LIN {X 0,Y 564.129,Z 608.975,A -85,B 0,C 180,E1 27064.074,E2 27064.074} C_VEL
LIN {X 0,Y 564.426,Z 588.414,A -85,B 0,C 180,E1 27063.622,E2 27063.622} C_VEL
LIN {X 0,Y 565.706,Z 337.003,A -85,B 0,C 180,E1 27060.121,E2 27060.121} C_VEL
LIN {X 0,Y 564.243,Z 328.893,A -85,B 0,C 180,E1 27059.903,E2 27059.903} C_VEL
LIN {X 0,Y 565.2,Z 283.5,A -85,B 0,C 180,E1 27056.615,E2 27056.615} C_VEL
LIN {X 0,Y 565.283,Z 271.236,A -85,B 0,C 180,E1 27055.692,E2 27055.692} C_VEL
LIN {X 0,Y 560.332,Z 258.325,A -85,B 0,C 180,E1 27054.283,E2 27054.283} C_VEL
LIN {X 0,Y 560.259,Z 257.932,A -85,B 0,C 180,E1 27053.598,E2 27053.598} C_VEL
LIN {X 0,Y 560.276,Z 257.928,A -85,B 0,C 180,E1 27050.278,E2 27050.278} C_VEL
LIN {X 0,Y 560.273,Z 257.936,A -85,B 0,C 180,E1 27047.024,E2 27047.024} C_VEL
LIN {X 0,Y 560.266,Z 257.946,A -85,B 0,C 180,E1 27043.681,E2 27043.681} C_VEL
LIN {X 0,Y 560.273,Z 257.941,A -85,B 0,C 180,E1 27040.359,E2 27040.359} C_VEL
LIN {X 0,Y 560.265,Z 257.937,A -85,B 0,C 180,E1 27036.919,E2 27036.919} C_VEL
LIN {X 0,Y 560.273,Z 257.946,A -85,B 0,C 180,E1 27033.552,E2 27033.552} C_VEL
LIN {X 0,Y 560.267,Z 257.933,A -85,B 0,C 180,E1 27030.216,E2 27030.216} C_VEL
LIN {X 0,Y 560.256,Z 257.943,A -85,B 0,C 180,E1 27026.837,E2 27026.837} C_VEL
LIN {X 0,Y 560.279,Z 257.944,A -85,B 0,C 180,E1 27023.562,E2 27023.562} C_VEL
LIN {X 0,Y 560.246,Z 257.944,A -85,B 0,C 180,E1 27020.366,E2 27020.366} C_VEL
LIN {X 0,Y 560.263,Z 257.948,A -85,B 0,C 180,E1 27017.019,E2 27017.019} C_VEL
LIN {X 0,Y 560.28,Z 257.938,A -85,B 0,C 180,E1 27013.73,E2 27013.73} C_VEL
LIN {X 0,Y 560.233,Z 257.94,A -85,B 0,C 180,E1 27010.469,E2 27010.469} C_VEL
LIN {X 0,Y 560.274,Z 257.945,A -85,B 0,C 180,E1 27007.176,E2 27007.176} C_VEL
LIN {X 0,Y 560.24,Z 257.945,A -85,B 0,C 180,E1 27003.957,E2 27003.957} C_VEL
LIN {X 0,Y 560.224,Z 257.947,A -85,B 0,C 180,E1 27000.614,E2 27000.614} C_VEL
LIN {X 0,Y 560.278,Z 257.945,A -85,B 0,C 180,E1 26997.443,E2 26997.443} C_VEL
LIN {X 0,Y 560.21,Z 257.947,A -85,B 0,C 180,E1 26994.264,E2 26994.264} C_VEL
LIN {X 0,Y 560.256,Z 257.949,A -85,B 0,C 180,E1 26991.068,E2 26991.068} C_VEL
LIN {X 0,Y 560.209,Z 257.945,A -85,B 0,C 180,E1 26987.947,E2 26987.947} C_VEL
LIN {X 0,Y 560.203,Z 257.945,A -85,B 0,C 180,E1 26984.53,E2 26984.53} C_VEL
LIN {X 0,Y 560.246,Z 257.949,A -85,B 0,C 180,E1 26981.478,E2 26981.478} C_VEL
LIN {X 0,Y 560.206,Z 257.948,A -85,B 0,C 180,E1 26978.318,E2 26978.318} C_VEL
LIN {X 0,Y 560.277,Z 257.949,A -85,B 0,C 180,E1 26975.205,E2 26975.205} C_VEL
LIN {X 0,Y 560.214,Z 257.948,A -85,B 0,C 180,E1 26972.005,E2 26972.005} C_VEL
LIN {X 0,Y 560.248,Z 257.935,A -85,B 0,C 180,E1 26968.712,E2 26968.712} C_VEL
LIN {X 0,Y 560.249,Z 257.949,A -85,B 0,C 180,E1 26965.537,E2 26965.537} C_VEL
LIN {X 0,Y 560.229,Z 257.942,A -85,B 0,C 180,E1 26962.243,E2 26962.243} C_VEL
LIN {X 0,Y 560.283,Z 257.933,A -85,B 0,C 180,E1 26959.012,E2 26959.012} C_VEL
LIN {X 0,Y 560.241,Z 257.949,A -85,B 0,C 180,E1 26955.748,E2 26955.748} C_VEL
LIN {X 0,Y 560.252,Z 257.945,A -85,B 0,C 180,E1 26952.367,E2 26952.367} C_VEL
LIN {X 0,Y 560.281,Z 257.941,A -85,B 0,C 180,E1 26949.079,E2 26949.079} C_VEL
LIN {X 0,Y 560.319,Z 258.259,A -85,B 0,C 180,E1 26948.567,E2 26948.567} C_VEL
LIN {X 0,Y 564.336,Z 267.794,A -85,B 0,C 180,E1 26947.551,E2 26947.551} C_VEL
LIN {X 0,Y 566.828,Z 273.642,A -85,B 0,C 180,E1 26946.959,E2 26946.959} C_VEL
LIN {X 0,Y 566.291,Z 302.779,A -85,B 0,C 180,E1 26945.075,E2 26945.075} C_VEL
LIN {X 0,Y 567.756,Z 312.242,A -85,B 0,C 180,E1 26944.825,E2 26944.825} C_VEL
LIN {X 0,Y 566.415,Z 533.81,A -85,B 0,C 180,E1 26941.628,E2 26941.628} C_VEL
LIN {X 0,Y 565.943,Z 609.207,A -85,B 0,C 180,E1 26940.529,E2 26940.529} C_VEL
LIN {X 0,Y 565.546,Z 630.675,A -85,B 0,C 180,E1 26940.025,E2 26940.025} C_VEL
LIN {X 0,Y 565.085,Z 652.51,A -85,B 0,C 180,E1 26939.319,E2 26939.319} C_VEL
LIN {X 0,Y 564.579,Z 673.407,A -85,B 0,C 180,E1 26938.449,E2 26938.449} C_VEL
LIN {X 0,Y 563.935,Z 693.757,A -85,B 0,C 180,E1 26937.392,E2 26937.392} C_VEL
LIN {X 0,Y 563.301,Z 714.152,A -85,B 0,C 180,E1 26936.116,E2 26936.116} C_VEL
LIN {X 0,Y 562.7,Z 732.379,A -85,B 0,C 180,E1 26934.771,E2 26934.771} C_VEL
LIN {X 0,Y 562.102,Z 750.23,A -85,B 0,C 180,E1 26933.229,E2 26933.229} C_VEL
LIN {X 0,Y 561.572,Z 766.692,A -85,B 0,C 180,E1 26931.571,E2 26931.571} C_VEL
LIN {X 0,Y 561.082,Z 782.874,A -85,B 0,C 180,E1 26929.682,E2 26929.682} C_VEL
LIN {X 0,Y 560.714,Z 797.045,A -85,B 0,C 180,E1 26927.753,E2 26927.753} C_VEL
LIN {X 0,Y 560.417,Z 809.739,A -85,B 0,C 180,E1 26925.735,E2 26925.735} C_VEL
LIN {X 0,Y 560.198,Z 820.334,A -85,B 0,C 180,E1 26923.732,E2 26923.732} C_VEL
LIN {X 0,Y 560.057,Z 830.069,A -85,B 0,C 180,E1 26921.534,E2 26921.534} C_VEL
LIN {X 0,Y 559.982,Z 837.937,A -85,B 0,C 180,E1 26919.351,E2 26919.351} C_VEL
LIN {X 0,Y 559.938,Z 843.907,A -85,B 0,C 180,E1 26917.18,E2 26917.18} C_VEL
LIN {X 0,Y 559.917,Z 848.581,A -85,B 0,C 180,E1 26914.841,E2 26914.841} C_VEL
LIN {X 0,Y 559.907,Z 851.338,A -85,B 0,C 180,E1 26912.661,E2 26912.661} C_VEL
LIN {X 0,Y 559.896,Z 852.395,A -85,B 0,C 180,E1 26910.512,E2 26910.512} C_VEL
LIN {X 0,Y 559.901,Z 851.948,A -85,B 0,C 180,E1 26908.26,E2 26908.26} C_VEL
LIN {X 0,Y 559.908,Z 849.994,A -85,B 0,C 180,E1 26906.109,E2 26906.109} C_VEL
LIN {X 0,Y 559.921,Z 846.398,A -85,B 0,C 180,E1 26903.952,E2 26903.952} C_VEL
LIN {X 0,Y 559.958,Z 841.281,A -85,B 0,C 180,E1 26901.788,E2 26901.788} C_VEL
LIN {X 0,Y 560.01,Z 834.757,A -85,B 0,C 180,E1 26899.715,E2 26899.715} C_VEL
LIN {X 0,Y 560.11,Z 826.141,A -85,B 0,C 180,E1 26897.526,E2 26897.526} C_VEL
LIN {X 0,Y 560.286,Z 816.122,A -85,B 0,C 180,E1 26895.427,E2 26895.427} C_VEL
LIN {X 0,Y 560.527,Z 804.629,A -85,B 0,C 180,E1 26893.417,E2 26893.417} C_VEL
LIN {X 0,Y 560.838,Z 791.792,A -85,B 0,C 180,E1 26891.499,E2 26891.499} C_VEL
LIN {X 0,Y 561.233,Z 777.662,A -85,B 0,C 180,E1 26889.672,E2 26889.672} C_VEL
LIN {X 0,Y 561.73,Z 761.816,A -85,B 0,C 180,E1 26887.907,E2 26887.907} C_VEL
LIN {X 0,Y 562.275,Z 745.074,A -85,B 0,C 180,E1 26886.305,E2 26886.305} C_VEL
LIN {X 0,Y 562.893,Z 726.402,A -85,B 0,C 180,E1 26884.767,E2 26884.767} C_VEL
LIN {X 0,Y 563.512,Z 707.543,A -85,B 0,C 180,E1 26883.441,E2 26883.441} C_VEL
LIN {X 0,Y 564.132,Z 687.761,A -85,B 0,C 180,E1 26882.274,E2 26882.274} C_VEL
LIN {X 0,Y 564.706,Z 667.063,A -85,B 0,C 180,E1 26881.269,E2 26881.269} C_VEL
LIN {X 0,Y 565.266,Z 645.686,A -85,B 0,C 180,E1 26880.438,E2 26880.438} C_VEL
LIN {X 0,Y 565.67,Z 624.869,A -85,B 0,C 180,E1 26879.819,E2 26879.819} C_VEL
LIN {X 0,Y 565.988,Z 603.285,A -85,B 0,C 180,E1 26879.372,E2 26879.372} C_VEL
LIN {X 0,Y 567.374,Z 374.728,A -85,B 0,C 180,E1 26876.087,E2 26876.087} C_VEL
LIN {X 0,Y 567.577,Z 309.911,A -85,B 0,C 180,E1 26875.127,E2 26875.127} C_VEL
LIN {X 0,Y 566.208,Z 301.853,A -85,B 0,C 180,E1 26874.885,E2 26874.885} C_VEL
LIN {X 0,Y 566.754,Z 273.379,A -85,B 0,C 180,E1 26873.018,E2 26873.018} C_VEL
LIN {X 0,Y 560.335,Z 258.355,A -85,B 0,C 180,E1 26871.451,E2 26871.451} C_VEL
LIN {X 0,Y 560.279,Z 257.933,A -85,B 0,C 180,E1 26871.084,E2 26871.084} C_VEL
LIN {X 0,Y 560.242,Z 257.947,A -85,B 0,C 180,E1 26867.854,E2 26867.854} C_VEL
LIN {X 0,Y 560.254,Z 257.947,A -85,B 0,C 180,E1 26864.452,E2 26864.452} C_VEL
LIN {X 0,Y 560.283,Z 257.932,A -85,B 0,C 180,E1 26861.144,E2 26861.144} C_VEL
LIN {X 0,Y 560.228,Z 257.942,A -85,B 0,C 180,E1 26857.875,E2 26857.875} C_VEL
LIN {X 0,Y 560.263,Z 257.949,A -85,B 0,C 180,E1 26854.577,E2 26854.577} C_VEL
LIN {X 0,Y 560.237,Z 257.936,A -85,B 0,C 180,E1 26851.408,E2 26851.408} C_VEL
LIN {X 0,Y 560.221,Z 257.948,A -85,B 0,C 180,E1 26848.11,E2 26848.11} C_VEL
LIN {X 0,Y 560.272,Z 257.945,A -85,B 0,C 180,E1 26844.967,E2 26844.967} C_VEL
LIN {X 0,Y 560.207,Z 257.948,A -85,B 0,C 180,E1 26841.792,E2 26841.792} C_VEL
LIN {X 0,Y 560.265,Z 257.948,A -85,B 0,C 180,E1 26838.629,E2 26838.629} C_VEL
LIN {X 0,Y 560.2,Z 257.945,A -85,B 0,C 180,E1 26835.529,E2 26835.529} C_VEL
LIN {X 0,Y 560.213,Z 257.945,A -85,B 0,C 180,E1 26832.158,E2 26832.158} C_VEL
LIN {X 0,Y 560.228,Z 257.949,A -85,B 0,C 180,E1 26829.139,E2 26829.139} C_VEL
LIN {X 0,Y 560.209,Z 257.948,A -85,B 0,C 180,E1 26825.839,E2 26825.839} C_VEL
LIN {X 0,Y 560.278,Z 257.944,A -85,B 0,C 180,E1 26822.659,E2 26822.659} C_VEL
LIN {X 0,Y 560.216,Z 257.947,A -85,B 0,C 180,E1 26819.488,E2 26819.488} C_VEL
LIN {X 0,Y 560.255,Z 257.944,A -85,B 0,C 180,E1 26816.214,E2 26816.214} C_VEL
LIN {X 0,Y 560.247,Z 257.944,A -85,B 0,C 180,E1 26813.029,E2 26813.029} C_VEL
LIN {X 0,Y 560.23,Z 257.94,A -85,B 0,C 180,E1 26809.719,E2 26809.719} C_VEL
LIN {X 0,Y 560.284,Z 257.941,A -85,B 0,C 180,E1 26806.48,E2 26806.48} C_VEL
LIN {X 0,Y 560.238,Z 257.946,A -85,B 0,C 180,E1 26803.301,E2 26803.301} C_VEL
LIN {X 0,Y 560.262,Z 257.942,A -85,B 0,C 180,E1 26799.961,E2 26799.961} C_VEL
LIN {X 0,Y 560.28,Z 257.946,A -85,B 0,C 180,E1 26796.661,E2 26796.661} C_VEL
LIN {X 0,Y 560.28,Z 257.942,A -85,B 0,C 180,E1 26796.239,E2 26796.239} C_VEL
LIN {X 0,Y 559.29,Z 258.064,A -85,B 0,C 180,E1 26795.451,E2 26795.451} C_VEL
LIN {X 0,Y 552.863,Z 258.863,A -85,B 0,C 180,E1 26793.24,E2 26793.24} C_VEL
LIN {X 0,Y 552.339,Z 258.936,A -85,B 0,C 180,E1 26792.664,E2 26792.664} C_VEL
LIN {X 0,Y 552.312,Z 258.925,A -85,B 0,C 180,E1 26789.302,E2 26789.302} C_VEL
LIN {X 0,Y 552.339,Z 258.93,A -85,B 0,C 180,E1 26785.988,E2 26785.988} C_VEL
LIN {X 0,Y 552.336,Z 258.922,A -85,B 0,C 180,E1 26782.537,E2 26782.537} C_VEL
LIN {X 0,Y 552.321,Z 258.934,A -85,B 0,C 180,E1 26779.193,E2 26779.193} C_VEL
LIN {X 0,Y 552.342,Z 258.93,A -85,B 0,C 180,E1 26775.793,E2 26775.793} C_VEL
LIN {X 0,Y 552.33,Z 258.93,A -85,B 0,C 180,E1 26772.389,E2 26772.389} C_VEL
LIN {X 0,Y 552.328,Z 258.921,A -85,B 0,C 180,E1 26769.18,E2 26769.18} C_VEL
LIN {X 0,Y 552.355,Z 259.158,A -85,B 0,C 180,E1 26766.207,E2 26766.207} C_VEL
LIN {X 0,Y 554.368,Z 264.541,A -85,B 0,C 180,E1 26765.568,E2 26765.568} C_VEL
LIN {X 0,Y 558.48,Z 275.126,A -85,B 0,C 180,E1 26764.413,E2 26764.413} C_VEL
LIN {X 0,Y 557.294,Z 318.934,A -85,B 0,C 180,E1 26761.151,E2 26761.151} C_VEL
LIN {X 0,Y 557.128,Z 329.515,A -85,B 0,C 180,E1 26760.412,E2 26760.412} C_VEL
LIN {X 0,Y 558.767,Z 339.665,A -85,B 0,C 180,E1 26760.159,E2 26760.159} C_VEL
LIN {X 0,Y 557.241,Z 590.093,A -85,B 0,C 180,E1 26756.626,E2 26756.626} C_VEL
LIN {X 0,Y 556.889,Z 610.371,A -85,B 0,C 180,E1 26756.16,E2 26756.16} C_VEL
LIN {X 0,Y 556.454,Z 630.143,A -85,B 0,C 180,E1 26755.517,E2 26755.517} C_VEL
LIN {X 0,Y 555.93,Z 650.229,A -85,B 0,C 180,E1 26754.661,E2 26754.661} C_VEL
LIN {X 0,Y 555.374,Z 668.831,A -85,B 0,C 180,E1 26753.67,E2 26753.67} C_VEL
LIN {X 0,Y 554.772,Z 687.426,A -85,B 0,C 180,E1 26752.462,E2 26752.462} C_VEL
LIN {X 0,Y 554.193,Z 704.475,A -85,B 0,C 180,E1 26751.131,E2 26751.131} C_VEL
LIN {X 0,Y 553.647,Z 720.769,A -85,B 0,C 180,E1 26749.627,E2 26749.627} C_VEL
LIN {X 0,Y 553.165,Z 735.716,A -85,B 0,C 180,E1 26748.004,E2 26748.004} C_VEL
LIN {X 0,Y 552.773,Z 749.225,A -85,B 0,C 180,E1 26746.282,E2 26746.282} C_VEL
LIN {X 0,Y 552.443,Z 761.975,A -85,B 0,C 180,E1 26744.356,E2 26744.356} C_VEL
LIN {X 0,Y 552.224,Z 772.578,A -85,B 0,C 180,E1 26742.442,E2 26742.442} C_VEL
LIN {X 0,Y 552.074,Z 781.763,A -85,B 0,C 180,E1 26740.434,E2 26740.434} C_VEL
LIN {X 0,Y 551.983,Z 789.382,A -85,B 0,C 180,E1 26738.332,E2 26738.332} C_VEL
LIN {X 0,Y 551.934,Z 794.889,A -85,B 0,C 180,E1 26736.344,E2 26736.344} C_VEL
LIN {X 0,Y 551.917,Z 799.202,A -85,B 0,C 180,E1 26734.155,E2 26734.155} C_VEL
LIN {X 0,Y 551.914,Z 801.641,A -85,B 0,C 180,E1 26732.076,E2 26732.076} C_VEL
LIN {X 0,Y 551.914,Z 802.495,A -85,B 0,C 180,E1 26730,E2 26730} C_VEL
LIN {X 0,Y 551.909,Z 801.633,A -85,B 0,C 180,E1 26727.82,E2 26727.82} C_VEL
LIN {X 0,Y 551.914,Z 799.18,A -85,B 0,C 180,E1 26725.74,E2 26725.74} C_VEL
LIN {X 0,Y 551.932,Z 794.854,A -85,B 0,C 180,E1 26723.551,E2 26723.551} C_VEL
LIN {X 0,Y 551.983,Z 788.979,A -85,B 0,C 180,E1 26721.458,E2 26721.458} C_VEL
LIN {X 0,Y 552.075,Z 781.702,A -85,B 0,C 180,E1 26719.46,E2 26719.46} C_VEL
LIN {X 0,Y 552.228,Z 772.238,A -85,B 0,C 180,E1 26717.398,E2 26717.398} C_VEL
LIN {X 0,Y 552.451,Z 761.83,A -85,B 0,C 180,E1 26715.53,E2 26715.53} C_VEL
LIN {X 0,Y 552.774,Z 749.093,A -85,B 0,C 180,E1 26713.611,E2 26713.611} C_VEL
LIN {X 0,Y 553.196,Z 734.628,A -85,B 0,C 180,E1 26711.779,E2 26711.779} C_VEL
LIN {X 0,Y 553.707,Z 718.916,A -85,B 0,C 180,E1 26710.1,E2 26710.1} C_VEL
LIN {X 0,Y 554.284,Z 701.829,A -85,B 0,C 180,E1 26708.56,E2 26708.56} C_VEL
LIN {X 0,Y 554.885,Z 683.925,A -85,B 0,C 180,E1 26707.207,E2 26707.207} C_VEL
LIN {X 0,Y 555.472,Z 665.466,A -85,B 0,C 180,E1 26706.045,E2 26706.045} C_VEL
LIN {X 0,Y 556.05,Z 646.345,A -85,B 0,C 180,E1 26705.061,E2 26705.061} C_VEL
LIN {X 0,Y 556.56,Z 626.554,A -85,B 0,C 180,E1 26704.26,E2 26704.26} C_VEL
LIN {X 0,Y 556.951,Z 606.601,A -85,B 0,C 180,E1 26703.65,E2 26703.65} C_VEL
LIN {X 0,Y 557.269,Z 585.492,A -85,B 0,C 180,E1 26703.208,E2 26703.208} C_VEL
LIN {X 0,Y 558.743,Z 338.271,A -85,B 0,C 180,E1 26699.729,E2 26699.729} C_VEL
LIN {X 0,Y 557.057,Z 328.892,A -85,B 0,C 180,E1 26699.473,E2 26699.473} C_VEL
LIN {X 0,Y 558.187,Z 284.604,A -85,B 0,C 180,E1 26696.217,E2 26696.217} C_VEL
LIN {X 0,Y 558.38,Z 274.72,A -85,B 0,C 180,E1 26695.457,E2 26695.457} C_VEL
LIN {X 0,Y 552.364,Z 259.241,A -85,B 0,C 180,E1 26693.724,E2 26693.724} C_VEL
LIN {X 0,Y 552.336,Z 258.926,A -85,B 0,C 180,E1 26692.627,E2 26692.627} C_VEL
LIN {X 0,Y 552.343,Z 258.929,A -85,B 0,C 180,E1 26689.172,E2 26689.172} C_VEL
LIN {X 0,Y 552.325,Z 258.925,A -85,B 0,C 180,E1 26685.797,E2 26685.797} C_VEL
LIN {X 0,Y 552.329,Z 258.916,A -85,B 0,C 180,E1 26682.472,E2 26682.472} C_VEL
LIN {X 0,Y 552.334,Z 258.931,A -85,B 0,C 180,E1 26679.048,E2 26679.048} C_VEL
LIN {X 0,Y 552.333,Z 258.927,A -85,B 0,C 180,E1 26675.632,E2 26675.632} C_VEL
LIN {X 0,Y 552.328,Z 258.923,A -85,B 0,C 180,E1 26672.278,E2 26672.278} C_VEL
LIN {X 0,Y 552.319,Z 258.935,A -85,B 0,C 180,E1 26668.818,E2 26668.818} C_VEL
LIN {X 0,Y 552.339,Z 258.93,A -85,B 0,C 180,E1 26665.521,E2 26665.521} C_VEL
LIN {X 0,Y 552.316,Z 258.927,A -85,B 0,C 180,E1 26662.232,E2 26662.232} C_VEL
LIN {X 0,Y 552.309,Z 258.932,A -85,B 0,C 180,E1 26658.778,E2 26658.778} C_VEL
LIN {X 0,Y 552.345,Z 258.934,A -85,B 0,C 180,E1 26655.433,E2 26655.433} C_VEL
LIN {X 0,Y 552.306,Z 258.933,A -85,B 0,C 180,E1 26652.122,E2 26652.122} C_VEL
LIN {X 0,Y 552.298,Z 258.936,A -85,B 0,C 180,E1 26648.725,E2 26648.725} C_VEL
LIN {X 0,Y 552.343,Z 258.929,A -85,B 0,C 180,E1 26645.506,E2 26645.506} C_VEL
LIN {X 0,Y 552.284,Z 258.933,A -85,B 0,C 180,E1 26642.283,E2 26642.283} C_VEL
LIN {X 0,Y 552.31,Z 258.936,A -85,B 0,C 180,E1 26638.963,E2 26638.963} C_VEL
LIN {X 0,Y 552.294,Z 258.934,A -85,B 0,C 180,E1 26635.847,E2 26635.847} C_VEL
LIN {X 0,Y 552.272,Z 258.934,A -85,B 0,C 180,E1 26632.51,E2 26632.51} C_VEL
LIN {X 0,Y 552.33,Z 258.936,A -85,B 0,C 180,E1 26629.36,E2 26629.36} C_VEL
LIN {X 0,Y 552.26,Z 258.938,A -85,B 0,C 180,E1 26626.174,E2 26626.174} C_VEL
LIN {X 0,Y 552.296,Z 258.938,A -85,B 0,C 180,E1 26622.91,E2 26622.91} C_VEL
LIN {X 0,Y 552.279,Z 258.935,A -85,B 0,C 180,E1 26619.77,E2 26619.77} C_VEL
LIN {X 0,Y 552.273,Z 258.935,A -85,B 0,C 180,E1 26616.415,E2 26616.415} C_VEL
LIN {X 0,Y 552.342,Z 258.933,A -85,B 0,C 180,E1 26613.178,E2 26613.178} C_VEL
LIN {X 0,Y 552.279,Z 258.933,A -85,B 0,C 180,E1 26610.022,E2 26610.022} C_VEL
LIN {X 0,Y 552.317,Z 258.935,A -85,B 0,C 180,E1 26606.735,E2 26606.735} C_VEL
LIN {X 0,Y 552.306,Z 258.928,A -85,B 0,C 180,E1 26603.574,E2 26603.574} C_VEL
LIN {X 0,Y 552.296,Z 258.935,A -85,B 0,C 180,E1 26600.279,E2 26600.279} C_VEL
LIN {X 0,Y 552.345,Z 258.934,A -85,B 0,C 180,E1 26596.996,E2 26596.996} C_VEL
LIN {X 0,Y 552.302,Z 258.927,A -85,B 0,C 180,E1 26593.752,E2 26593.752} C_VEL
LIN {X 0,Y 552.314,Z 258.924,A -85,B 0,C 180,E1 26590.347,E2 26590.347} C_VEL
LIN {X 0,Y 552.38,Z 259.179,A -85,B 0,C 180,E1 26589.176,E2 26589.176} C_VEL
LIN {X 0,Y 554.318,Z 264.07,A -85,B 0,C 180,E1 26588.615,E2 26588.615} C_VEL
LIN {X 0,Y 560.022,Z 277.103,A -85,B 0,C 180,E1 26587.245,E2 26587.245} C_VEL
LIN {X 0,Y 559.467,Z 302.819,A -85,B 0,C 180,E1 26585.567,E2 26585.567} C_VEL
LIN {X 0,Y 561.178,Z 313.62,A -85,B 0,C 180,E1 26585.273,E2 26585.273} C_VEL
LIN {X 0,Y 559.597,Z 534.701,A -85,B 0,C 180,E1 26582.046,E2 26582.046} C_VEL
LIN {X 0,Y 559.047,Z 609.207,A -85,B 0,C 180,E1 26580.946,E2 26580.946} C_VEL
LIN {X 0,Y 558.581,Z 630.676,A -85,B 0,C 180,E1 26580.438,E2 26580.438} C_VEL
LIN {X 0,Y 558.051,Z 652.58,A -85,B 0,C 180,E1 26579.722,E2 26579.722} C_VEL
LIN {X 0,Y 557.44,Z 673.407,A -85,B 0,C 180,E1 26578.848,E2 26578.848} C_VEL
LIN {X 0,Y 556.703,Z 693.759,A -85,B 0,C 180,E1 26577.779,E2 26577.779} C_VEL
LIN {X 0,Y 555.951,Z 714.153,A -85,B 0,C 180,E1 26576.488,E2 26576.488} C_VEL
LIN {X 0,Y 555.199,Z 733.16,A -85,B 0,C 180,E1 26575.062,E2 26575.062} C_VEL
LIN {X 0,Y 554.505,Z 751.116,A -85,B 0,C 180,E1 26573.484,E2 26573.484} C_VEL
LIN {X 0,Y 553.868,Z 767.704,A -85,B 0,C 180,E1 26571.775,E2 26571.775} C_VEL
LIN {X 0,Y 553.323,Z 782.875,A -85,B 0,C 180,E1 26569.969,E2 26569.969} C_VEL
LIN {X 0,Y 552.873,Z 797.046,A -85,B 0,C 180,E1 26568.013,E2 26568.013} C_VEL
LIN {X 0,Y 552.515,Z 809.737,A -85,B 0,C 180,E1 26565.966,E2 26565.966} C_VEL
LIN {X 0,Y 552.258,Z 820.335,A -85,B 0,C 180,E1 26563.933,E2 26563.933} C_VEL
LIN {X 0,Y 552.085,Z 830.07,A -85,B 0,C 180,E1 26561.703,E2 26561.703} C_VEL
LIN {X 0,Y 551.99,Z 837.937,A -85,B 0,C 180,E1 26559.487,E2 26559.487} C_VEL
LIN {X 0,Y 551.939,Z 843.908,A -85,B 0,C 180,E1 26557.285,E2 26557.285} C_VEL
LIN {X 0,Y 551.92,Z 848.464,A -85,B 0,C 180,E1 26554.988,E2 26554.988} C_VEL
LIN {X 0,Y 551.909,Z 851.234,A -85,B 0,C 180,E1 26552.804,E2 26552.804} C_VEL
LIN {X 0,Y 551.898,Z 852.373,A -85,B 0,C 180,E1 26550.623,E2 26550.623} C_VEL
LIN {X 0,Y 551.899,Z 852.015,A -85,B 0,C 180,E1 26548.339,E2 26548.339} C_VEL
LIN {X 0,Y 551.904,Z 850.221,A -85,B 0,C 180,E1 26546.261,E2 26546.261} C_VEL
LIN {X 0,Y 551.922,Z 846.603,A -85,B 0,C 180,E1 26543.969,E2 26543.969} C_VEL
LIN {X 0,Y 551.965,Z 841.584,A -85,B 0,C 180,E1 26541.773,E2 26541.773} C_VEL
LIN {X 0,Y 552.025,Z 835.112,A -85,B 0,C 180,E1 26539.67,E2 26539.67} C_VEL
LIN {X 0,Y 552.147,Z 826.537,A -85,B 0,C 180,E1 26537.434,E2 26537.434} C_VEL
LIN {X 0,Y 552.351,Z 816.69,A -85,B 0,C 180,E1 26535.32,E2 26535.32} C_VEL
LIN {X 0,Y 552.633,Z 805.272,A -85,B 0,C 180,E1 26533.282,E2 26533.282} C_VEL
LIN {X 0,Y 553.028,Z 791.794,A -85,B 0,C 180,E1 26531.228,E2 26531.228} C_VEL
LIN {X 0,Y 553.514,Z 777.375,A -85,B 0,C 180,E1 26529.342,E2 26529.342} C_VEL
LIN {X 0,Y 554.097,Z 761.625,A -85,B 0,C 180,E1 26527.565,E2 26527.565} C_VEL
LIN {X 0,Y 554.754,Z 744.464,A -85,B 0,C 180,E1 26525.907,E2 26525.907} C_VEL
LIN {X 0,Y 555.498,Z 725.678,A -85,B 0,C 180,E1 26524.35,E2 26524.35} C_VEL
LIN {X 0,Y 556.241,Z 706.421,A -85,B 0,C 180,E1 26522.993,E2 26522.993} C_VEL
LIN {X 0,Y 556.971,Z 686.522,A -85,B 0,C 180,E1 26521.815,E2 26521.815} C_VEL
LIN {X 0,Y 557.64,Z 666.234,A -85,B 0,C 180,E1 26520.832,E2 26520.832} C_VEL
LIN {X 0,Y 558.264,Z 644.481,A -85,B 0,C 180,E1 26519.988,E2 26519.988} C_VEL
LIN {X 0,Y 558.791,Z 623.167,A -85,B 0,C 180,E1 26519.36,E2 26519.36} C_VEL
LIN {X 0,Y 559.113,Z 601.498,A -85,B 0,C 180,E1 26518.923,E2 26518.923} C_VEL
LIN {X 0,Y 560.716,Z 377.149,A -85,B 0,C 180,E1 26515.665,E2 26515.665} C_VEL
LIN {X 0,Y 561.004,Z 311.391,A -85,B 0,C 180,E1 26514.68,E2 26514.68} C_VEL
LIN {X 0,Y 559.388,Z 302.303,A -85,B 0,C 180,E1 26514.417,E2 26514.417} C_VEL
LIN {X 0,Y 559.891,Z 276.6,A -85,B 0,C 180,E1 26512.71,E2 26512.71} C_VEL
LIN {X 0,Y 552.401,Z 259.313,A -85,B 0,C 180,E1 26510.854,E2 26510.854} C_VEL
LIN {X 0,Y 552.309,Z 258.936,A -85,B 0,C 180,E1 26510.281,E2 26510.281} C_VEL
LIN {X 0,Y 552.343,Z 258.935,A -85,B 0,C 180,E1 26506.966,E2 26506.966} C_VEL
LIN {X 0,Y 552.302,Z 258.936,A -85,B 0,C 180,E1 26503.753,E2 26503.753} C_VEL
LIN {X 0,Y 552.306,Z 258.937,A -85,B 0,C 180,E1 26500.348,E2 26500.348} C_VEL
LIN {X 0,Y 552.343,Z 258.922,A -85,B 0,C 180,E1 26497.07,E2 26497.07} C_VEL
LIN {X 0,Y 552.286,Z 258.936,A -85,B 0,C 180,E1 26493.804,E2 26493.804} C_VEL
LIN {X 0,Y 552.308,Z 258.929,A -85,B 0,C 180,E1 26490.457,E2 26490.457} C_VEL
LIN {X 0,Y 552.295,Z 258.936,A -85,B 0,C 180,E1 26487.376,E2 26487.376} C_VEL
LIN {X 0,Y 552.274,Z 258.936,A -85,B 0,C 180,E1 26484.038,E2 26484.038} C_VEL
LIN {X 0,Y 552.334,Z 258.936,A -85,B 0,C 180,E1 26480.892,E2 26480.892} C_VEL
LIN {X 0,Y 552.261,Z 258.938,A -85,B 0,C 180,E1 26477.707,E2 26477.707} C_VEL
LIN {X 0,Y 552.303,Z 258.938,A -85,B 0,C 180,E1 26474.467,E2 26474.467} C_VEL
LIN {X 0,Y 552.268,Z 258.934,A -85,B 0,C 180,E1 26471.381,E2 26471.381} C_VEL
LIN {X 0,Y 552.273,Z 258.934,A -85,B 0,C 180,E1 26467.993,E2 26467.993} C_VEL
LIN {X 0,Y 552.32,Z 258.938,A -85,B 0,C 180,E1 26464.881,E2 26464.881} C_VEL
LIN {X 0,Y 552.273,Z 258.935,A -85,B 0,C 180,E1 26461.66,E2 26461.66} C_VEL
LIN {X 0,Y 552.337,Z 258.931,A -85,B 0,C 180,E1 26458.444,E2 26458.444} C_VEL
LIN {X 0,Y 552.293,Z 258.937,A -85,B 0,C 180,E1 26455.223,E2 26455.223} C_VEL
LIN {X 0,Y 552.292,Z 258.934,A -85,B 0,C 180,E1 26451.777,E2 26451.777} C_VEL
LIN {X 0,Y 552.344,Z 258.935,A -85,B 0,C 180,E1 26448.514,E2 26448.514} C_VEL
LIN {X 0,Y 552.3,Z 258.932,A -85,B 0,C 180,E1 26445.211,E2 26445.211} C_VEL
LIN {X 0,Y 552.306,Z 258.929,A -85,B 0,C 180,E1 26441.748,E2 26441.748} C_VEL
LIN {X 0,Y 552.342,Z 258.93,A -85,B 0,C 180,E1 26438.44,E2 26438.44} C_VEL
LIN {X 0,Y 552.315,Z 258.936,A -85,B 0,C 180,E1 26435.085,E2 26435.085} C_VEL
LIN {X 0,Y 552.339,Z 258.936,A -85,B 0,C 180,E1 26432.664,E2 26432.664} C_VEL
LIN {X 0,Y 551.351,Z 259.069,A -85,B 0,C 180,E1 26431.865,E2 26431.865} C_VEL
LIN {X 0,Y 544.892,Z 259.852,A -85,B 0,C 180,E1 26429.621,E2 26429.621} C_VEL
LIN {X 0,Y 544.381,Z 259.909,A -85,B 0,C 180,E1 26429.036,E2 26429.036} C_VEL
LIN {X 0,Y 544.383,Z 259.921,A -85,B 0,C 180,E1 26425.549,E2 26425.549} C_VEL
LIN {X 0,Y 544.397,Z 259.911,A -85,B 0,C 180,E1 26422.16,E2 26422.16} C_VEL
LIN {X 0,Y 544.403,Z 259.913,A -85,B 0,C 180,E1 26418.69,E2 26418.69} C_VEL
LIN {X 0,Y 544.387,Z 259.923,A -85,B 0,C 180,E1 26415.296,E2 26415.296} C_VEL
LIN {X 0,Y 544.392,Z 259.923,A -85,B 0,C 180,E1 26411.94,E2 26411.94} C_VEL
LIN {X 0,Y 544.393,Z 259.918,A -85,B 0,C 180,E1 26408.507,E2 26408.507} C_VEL
LIN {X 0,Y 544.429,Z 260.124,A -85,B 0,C 180,E1 26406.776,E2 26406.776} C_VEL
LIN {X 0,Y 546.9,Z 266.49,A -85,B 0,C 180,E1 26406.002,E2 26406.002} C_VEL
LIN {X 0,Y 551.518,Z 278.593,A -85,B 0,C 180,E1 26404.663,E2 26404.663} C_VEL
LIN {X 0,Y 550.088,Z 321.904,A -85,B 0,C 180,E1 26401.382,E2 26401.382} C_VEL
LIN {X 0,Y 549.978,Z 329.548,A -85,B 0,C 180,E1 26400.851,E2 26400.851} C_VEL
LIN {X 0,Y 551.844,Z 341.053,A -85,B 0,C 180,E1 26400.558,E2 26400.558} C_VEL
LIN {X 0,Y 550.091,Z 589.816,A -85,B 0,C 180,E1 26397.006,E2 26397.006} C_VEL
LIN {X 0,Y 549.687,Z 610.241,A -85,B 0,C 180,E1 26396.533,E2 26396.533} C_VEL
LIN {X 0,Y 549.193,Z 630.159,A -85,B 0,C 180,E1 26395.879,E2 26395.879} C_VEL
LIN {X 0,Y 548.585,Z 650.241,A -85,B 0,C 180,E1 26395.014,E2 26395.014} C_VEL
LIN {X 0,Y 547.939,Z 668.839,A -85,B 0,C 180,E1 26394.011,E2 26394.011} C_VEL
LIN {X 0,Y 547.252,Z 687.434,A -85,B 0,C 180,E1 26392.788,E2 26392.788} C_VEL
LIN {X 0,Y 546.545,Z 705.568,A -85,B 0,C 180,E1 26391.349,E2 26391.349} C_VEL
LIN {X 0,Y 545.91,Z 721.881,A -85,B 0,C 180,E1 26389.805,E2 26389.805} C_VEL
LIN {X 0,Y 545.354,Z 736.646,A -85,B 0,C 180,E1 26388.16,E2 26388.16} C_VEL
LIN {X 0,Y 544.901,Z 750.001,A -85,B 0,C 180,E1 26386.414,E2 26386.414} C_VEL
LIN {X 0,Y 544.522,Z 762.619,A -85,B 0,C 180,E1 26384.461,E2 26384.461} C_VEL
LIN {X 0,Y 544.256,Z 773.618,A -85,B 0,C 180,E1 26382.412,E2 26382.412} C_VEL
LIN {X 0,Y 544.086,Z 782.58,A -85,B 0,C 180,E1 26380.375,E2 26380.375} C_VEL
LIN {X 0,Y 543.992,Z 789.737,A -85,B 0,C 180,E1 26378.349,E2 26378.349} C_VEL
LIN {X 0,Y 543.937,Z 795.398,A -85,B 0,C 180,E1 26376.226,E2 26376.226} C_VEL
LIN {X 0,Y 543.918,Z 799.362,A -85,B 0,C 180,E1 26374.111,E2 26374.111} C_VEL
LIN {X 0,Y 543.914,Z 801.777,A -85,B 0,C 180,E1 26371.896,E2 26371.896} C_VEL
LIN {X 0,Y 543.908,Z 802.47,A -85,B 0,C 180,E1 26369.789,E2 26369.789} C_VEL
LIN {X 0,Y 543.905,Z 801.564,A -85,B 0,C 180,E1 26367.682,E2 26367.682} C_VEL
LIN {X 0,Y 543.913,Z 799.019,A -85,B 0,C 180,E1 26365.572,E2 26365.572} C_VEL
LIN {X 0,Y 543.937,Z 794.852,A -85,B 0,C 180,E1 26363.456,E2 26363.456} C_VEL
LIN {X 0,Y 543.995,Z 788.977,A -85,B 0,C 180,E1 26361.332,E2 26361.332} C_VEL
LIN {X 0,Y 544.101,Z 781.699,A -85,B 0,C 180,E1 26359.304,E2 26359.304} C_VEL
LIN {X 0,Y 544.276,Z 772.495,A -85,B 0,C 180,E1 26357.265,E2 26357.265} C_VEL
LIN {X 0,Y 544.547,Z 761.87,A -85,B 0,C 180,E1 26355.322,E2 26355.322} C_VEL
LIN {X 0,Y 544.904,Z 749.861,A -85,B 0,C 180,E1 26353.477,E2 26353.477} C_VEL
LIN {X 0,Y 545.36,Z 736.476,A -85,B 0,C 180,E1 26351.73,E2 26351.73} C_VEL
LIN {X 0,Y 545.916,Z 721.674,A -85,B 0,C 180,E1 26350.083,E2 26350.083} C_VEL
LIN {X 0,Y 546.554,Z 705.31,A -85,B 0,C 180,E1 26348.539,E2 26348.539} C_VEL
LIN {X 0,Y 547.229,Z 687.86,A -85,B 0,C 180,E1 26347.154,E2 26347.154} C_VEL
LIN {X 0,Y 547.889,Z 670.252,A -85,B 0,C 180,E1 26345.987,E2 26345.987} C_VEL
LIN {X 0,Y 548.555,Z 651.201,A -85,B 0,C 180,E1 26344.944,E2 26344.944} C_VEL
LIN {X 0,Y 549.165,Z 631.058,A -85,B 0,C 180,E1 26344.064,E2 26344.064} C_VEL
LIN {X 0,Y 549.679,Z 610.877,A -85,B 0,C 180,E1 26343.394,E2 26343.394} C_VEL
LIN {X 0,Y 550.088,Z 590.365,A -85,B 0,C 180,E1 26342.913,E2 26342.913} C_VEL
LIN {X 0,Y 551.847,Z 339.753,A -85,B 0,C 180,E1 26339.333,E2 26339.333} C_VEL
LIN {X 0,Y 549.904,Z 328.89,A -85,B 0,C 180,E1 26339.033,E2 26339.033} C_VEL
LIN {X 0,Y 551.247,Z 286.364,A -85,B 0,C 180,E1 26335.844,E2 26335.844} C_VEL
LIN {X 0,Y 551.485,Z 278.251,A -85,B 0,C 180,E1 26335.216,E2 26335.216} C_VEL
LIN {X 0,Y 545.423,Z 262.98,A -85,B 0,C 180,E1 26333.5,E2 26333.5} C_VEL
LIN {X 0,Y 544.437,Z 260.166,A -85,B 0,C 180,E1 26333.147,E2 26333.147} C_VEL
LIN {X 0,Y 544.381,Z 259.908,A -85,B 0,C 180,E1 26329.824,E2 26329.824} C_VEL
LIN {X 0,Y 544.397,Z 259.908,A -85,B 0,C 180,E1 26326.471,E2 26326.471} C_VEL
LIN {X 0,Y 544.395,Z 259.909,A -85,B 0,C 180,E1 26323.033,E2 26323.033} C_VEL
LIN {X 0,Y 544.391,Z 259.923,A -85,B 0,C 180,E1 26319.688,E2 26319.688} C_VEL
LIN {X 0,Y 544.389,Z 259.912,A -85,B 0,C 180,E1 26316.388,E2 26316.388} C_VEL
LIN {X 0,Y 544.386,Z 259.916,A -85,B 0,C 180,E1 26312.93,E2 26312.93} C_VEL
LIN {X 0,Y 544.396,Z 259.913,A -85,B 0,C 180,E1 26309.608,E2 26309.608} C_VEL
LIN {X 0,Y 544.381,Z 259.916,A -85,B 0,C 180,E1 26306.273,E2 26306.273} C_VEL
LIN {X 0,Y 544.374,Z 259.92,A -85,B 0,C 180,E1 26302.802,E2 26302.802} C_VEL
LIN {X 0,Y 544.404,Z 259.924,A -85,B 0,C 180,E1 26299.416,E2 26299.416} C_VEL
LIN {X 0,Y 544.374,Z 259.921,A -85,B 0,C 180,E1 26296.102,E2 26296.102} C_VEL
LIN {X 0,Y 544.363,Z 259.925,A -85,B 0,C 180,E1 26292.733,E2 26292.733} C_VEL
LIN {X 0,Y 544.406,Z 259.917,A -85,B 0,C 180,E1 26289.408,E2 26289.408} C_VEL
LIN {X 0,Y 544.358,Z 259.918,A -85,B 0,C 180,E1 26286.116,E2 26286.116} C_VEL
LIN {X 0,Y 544.35,Z 259.923,A -85,B 0,C 180,E1 26282.632,E2 26282.632} C_VEL
LIN {X 0,Y 544.408,Z 259.923,A -85,B 0,C 180,E1 26279.369,E2 26279.369} C_VEL
LIN {X 0,Y 544.34,Z 259.923,A -85,B 0,C 180,E1 26276.103,E2 26276.103} C_VEL
LIN {X 0,Y 544.342,Z 259.923,A -85,B 0,C 180,E1 26272.682,E2 26272.682} C_VEL
LIN {X 0,Y 544.374,Z 259.926,A -85,B 0,C 180,E1 26269.524,E2 26269.524} C_VEL
LIN {X 0,Y 544.321,Z 259.927,A -85,B 0,C 180,E1 26266.293,E2 26266.293} C_VEL
LIN {X 0,Y 544.382,Z 259.927,A -85,B 0,C 180,E1 26263.114,E2 26263.114} C_VEL
LIN {X 0,Y 544.332,Z 259.923,A -85,B 0,C 180,E1 26259.91,E2 26259.91} C_VEL
LIN {X 0,Y 544.335,Z 259.924,A -85,B 0,C 180,E1 26256.428,E2 26256.428} C_VEL
LIN {X 0,Y 544.401,Z 259.921,A -85,B 0,C 180,E1 26253.198,E2 26253.198} C_VEL
LIN {X 0,Y 544.34,Z 259.921,A -85,B 0,C 180,E1 26250.026,E2 26250.026} C_VEL
LIN {X 0,Y 544.374,Z 259.924,A -85,B 0,C 180,E1 26246.687,E2 26246.687} C_VEL
LIN {X 0,Y 544.374,Z 259.913,A -85,B 0,C 180,E1 26243.481,E2 26243.481} C_VEL
LIN {X 0,Y 544.353,Z 259.925,A -85,B 0,C 180,E1 26240.131,E2 26240.131} C_VEL
LIN {X 0,Y 544.401,Z 259.924,A -85,B 0,C 180,E1 26236.812,E2 26236.812} C_VEL
LIN {X 0,Y 544.379,Z 259.916,A -85,B 0,C 180,E1 26233.49,E2 26233.49} C_VEL
LIN {X 0,Y 544.366,Z 259.914,A -85,B 0,C 180,E1 26230.142,E2 26230.142} C_VEL
LIN {X 0,Y 544.419,Z 260.263,A -85,B 0,C 180,E1 26229.745,E2 26229.745} C_VEL
LIN {X 0,Y 547.095,Z 266.589,A -85,B 0,C 180,E1 26229.039,E2 26229.039} C_VEL
LIN {X 0,Y 553.22,Z 280.827,A -85,B 0,C 180,E1 26227.521,E2 26227.521} C_VEL
LIN {X 0,Y 552.676,Z 302.812,A -85,B 0,C 180,E1 26226.073,E2 26226.073} C_VEL
LIN {X 0,Y 554.633,Z 315.095,A -85,B 0,C 180,E1 26225.729,E2 26225.729} C_VEL
LIN {X 0,Y 552.81,Z 535.591,A -85,B 0,C 180,E1 26222.474,E2 26222.474} C_VEL
LIN {X 0,Y 552.178,Z 609.406,A -85,B 0,C 180,E1 26221.371,E2 26221.371} C_VEL
LIN {X 0,Y 551.642,Z 631.066,A -85,B 0,C 180,E1 26220.851,E2 26220.851} C_VEL
LIN {X 0,Y 551.021,Z 653.243,A -85,B 0,C 180,E1 26220.113,E2 26220.113} C_VEL
LIN {X 0,Y 550.33,Z 673.406,A -85,B 0,C 180,E1 26219.256,E2 26219.256} C_VEL
LIN {X 0,Y 549.499,Z 693.762,A -85,B 0,C 180,E1 26218.175,E2 26218.175} C_VEL
LIN {X 0,Y 548.622,Z 714.149,A -85,B 0,C 180,E1 26216.87,E2 26216.87} C_VEL
LIN {X 0,Y 547.764,Z 732.871,A -85,B 0,C 180,E1 26215.451,E2 26215.451} C_VEL
LIN {X 0,Y 546.98,Z 750.514,A -85,B 0,C 180,E1 26213.884,E2 26213.884} C_VEL
LIN {X 0,Y 546.249,Z 766.691,A -85,B 0,C 180,E1 26212.208,E2 26212.208} C_VEL
LIN {X 0,Y 545.572,Z 782.876,A -85,B 0,C 180,E1 26210.265,E2 26210.265} C_VEL
LIN {X 0,Y 545.042,Z 797.048,A -85,B 0,C 180,E1 26208.281,E2 26208.281} C_VEL
LIN {X 0,Y 544.625,Z 809.736,A -85,B 0,C 180,E1 26206.203,E2 26206.203} C_VEL
LIN {X 0,Y 544.321,Z 820.53,A -85,B 0,C 180,E1 26204.1,E2 26204.1} C_VEL
LIN {X 0,Y 544.119,Z 830.07,A -85,B 0,C 180,E1 26201.876,E2 26201.876} C_VEL
LIN {X 0,Y 544.002,Z 837.937,A -85,B 0,C 180,E1 26199.628,E2 26199.628} C_VEL
LIN {X 0,Y 543.941,Z 843.908,A -85,B 0,C 180,E1 26197.393,E2 26197.393} C_VEL
LIN {X 0,Y 543.921,Z 848.464,A -85,B 0,C 180,E1 26195.062,E2 26195.062} C_VEL
LIN {X 0,Y 543.911,Z 851.234,A -85,B 0,C 180,E1 26192.845,E2 26192.845} C_VEL
LIN {X 0,Y 543.898,Z 852.373,A -85,B 0,C 180,E1 26190.632,E2 26190.632} C_VEL
LIN {X 0,Y 543.899,Z 852.015,A -85,B 0,C 180,E1 26188.315,E2 26188.315} C_VEL
LIN {X 0,Y 543.905,Z 850.22,A -85,B 0,C 180,E1 26186.206,E2 26186.206} C_VEL
LIN {X 0,Y 543.925,Z 846.604,A -85,B 0,C 180,E1 26183.88,E2 26183.88} C_VEL
LIN {X 0,Y 543.965,Z 841.584,A -85,B 0,C 180,E1 26181.651,E2 26181.651} C_VEL
LIN {X 0,Y 544.042,Z 835.037,A -85,B 0,C 180,E1 26179.494,E2 26179.494} C_VEL
LIN {X 0,Y 544.195,Z 826.142,A -85,B 0,C 180,E1 26177.155,E2 26177.155} C_VEL
LIN {X 0,Y 544.438,Z 816.119,A -85,B 0,C 180,E1 26174.993,E2 26174.993} C_VEL
LIN {X 0,Y 544.779,Z 804.632,A -85,B 0,C 180,E1 26172.924,E2 26172.924} C_VEL
LIN {X 0,Y 545.232,Z 791.795,A -85,B 0,C 180,E1 26170.949,E2 26170.949} C_VEL
LIN {X 0,Y 545.792,Z 777.66,A -85,B 0,C 180,E1 26169.071,E2 26169.071} C_VEL
LIN {X 0,Y 546.482,Z 761.665,A -85,B 0,C 180,E1 26167.239,E2 26167.239} C_VEL
LIN {X 0,Y 547.231,Z 744.461,A -85,B 0,C 180,E1 26165.554,E2 26165.554} C_VEL
LIN {X 0,Y 548.102,Z 725.678,A -85,B 0,C 180,E1 26163.978,E2 26163.978} C_VEL
LIN {X 0,Y 548.959,Z 706.659,A -85,B 0,C 180,E1 26162.62,E2 26162.62} C_VEL
LIN {X 0,Y 549.786,Z 686.75,A -85,B 0,C 180,E1 26161.426,E2 26161.426} C_VEL
LIN {X 0,Y 550.55,Z 666.851,A -85,B 0,C 180,E1 26160.448,E2 26160.448} C_VEL
LIN {X 0,Y 551.26,Z 645.669,A -85,B 0,C 180,E1 26159.608,E2 26159.608} C_VEL
LIN {X 0,Y 551.83,Z 624.821,A -85,B 0,C 180,E1 26158.979,E2 26158.979} C_VEL
LIN {X 0,Y 552.242,Z 603.032,A -85,B 0,C 180,E1 26158.52,E2 26158.52} C_VEL
LIN {X 0,Y 554.097,Z 378.698,A -85,B 0,C 180,E1 26155.22,E2 26155.22} C_VEL
LIN {X 0,Y 554.465,Z 312.893,A -85,B 0,C 180,E1 26154.224,E2 26154.224} C_VEL
LIN {X 0,Y 552.591,Z 301.869,A -85,B 0,C 180,E1 26153.886,E2 26153.886} C_VEL
LIN {X 0,Y 553.141,Z 280.251,A -85,B 0,C 180,E1 26152.432,E2 26152.432} C_VEL
LIN {X 0,Y 545.255,Z 262.686,A -85,B 0,C 180,E1 26150.534,E2 26150.534} C_VEL
LIN {X 0,Y 544.396,Z 260.128,A -85,B 0,C 180,E1 26150.222,E2 26150.222} C_VEL
LIN {X 0,Y 544.404,Z 259.925,A -85,B 0,C 180,E1 26147.05,E2 26147.05} C_VEL
LIN {X 0,Y 544.362,Z 259.925,A -85,B 0,C 180,E1 26143.795,E2 26143.795} C_VEL
LIN {X 0,Y 544.366,Z 259.924,A -85,B 0,C 180,E1 26140.339,E2 26140.339} C_VEL
LIN {X 0,Y 544.405,Z 259.908,A -85,B 0,C 180,E1 26137.042,E2 26137.042} C_VEL
LIN {X 0,Y 544.347,Z 259.925,A -85,B 0,C 180,E1 26133.817,E2 26133.817} C_VEL
LIN {X 0,Y 544.369,Z 259.915,A -85,B 0,C 180,E1 26130.46,E2 26130.46} C_VEL
LIN {X 0,Y 544.36,Z 259.925,A -85,B 0,C 180,E1 26127.335,E2 26127.335} C_VEL
LIN {X 0,Y 544.337,Z 259.925,A -85,B 0,C 180,E1 26124.065,E2 26124.065} C_VEL
LIN {X 0,Y 544.396,Z 259.925,A -85,B 0,C 180,E1 26120.873,E2 26120.873} C_VEL
LIN {X 0,Y 544.324,Z 259.927,A -85,B 0,C 180,E1 26117.643,E2 26117.643} C_VEL
LIN {X 0,Y 544.352,Z 259.927,A -85,B 0,C 180,E1 26114.357,E2 26114.357} C_VEL
LIN {X 0,Y 544.34,Z 259.922,A -85,B 0,C 180,E1 26111.227,E2 26111.227} C_VEL
LIN {X 0,Y 544.33,Z 259.923,A -85,B 0,C 180,E1 26107.918,E2 26107.918} C_VEL
LIN {X 0,Y 544.394,Z 259.927,A -85,B 0,C 180,E1 26104.741,E2 26104.741} C_VEL
LIN {X 0,Y 544.336,Z 259.925,A -85,B 0,C 180,E1 26101.473,E2 26101.473} C_VEL
LIN {X 0,Y 544.372,Z 259.921,A -85,B 0,C 180,E1 26098.21,E2 26098.21} C_VEL
LIN {X 0,Y 544.377,Z 259.926,A -85,B 0,C 180,E1 26094.942,E2 26094.942} C_VEL
LIN {X 0,Y 544.35,Z 259.924,A -85,B 0,C 180,E1 26091.656,E2 26091.656} C_VEL
LIN {X 0,Y 544.402,Z 259.921,A -85,B 0,C 180,E1 26088.344,E2 26088.344} C_VEL
LIN {X 0,Y 544.373,Z 259.92,A -85,B 0,C 180,E1 26085.035,E2 26085.035} C_VEL
LIN {X 0,Y 544.365,Z 259.918,A -85,B 0,C 180,E1 26081.694,E2 26081.694} C_VEL
LIN {X 0,Y 544.404,Z 259.918,A -85,B 0,C 180,E1 26078.449,E2 26078.449} C_VEL
LIN {X 0,Y 544.374,Z 259.925,A -85,B 0,C 180,E1 26075.127,E2 26075.127} C_VEL
LIN {X 0,Y 544.381,Z 259.92,A -85,B 0,C 180,E1 26071.714,E2 26071.714} C_VEL
LIN {X 0,Y 544.381,Z 259.909,A -85,B 0,C 180,E1 26069.036,E2 26069.036} C_VEL
LIN {X 0,Y 543.423,Z 260.03,A -85,B 0,C 180,E1 26068.225,E2 26068.225} C_VEL
LIN {X 0,Y 536.888,Z 260.857,A -85,B 0,C 180,E1 26065.889,E2 26065.889} C_VEL
LIN {X 0,Y 536.44,Z 260.912,A -85,B 0,C 180,E1 26065.355,E2 26065.355} C_VEL
LIN {X 0,Y 536.465,Z 260.901,A -85,B 0,C 180,E1 26061.909,E2 26061.909} C_VEL
LIN {X 0,Y 536.457,Z 260.896,A -85,B 0,C 180,E1 26058.431,E2 26058.431} C_VEL
LIN {X 0,Y 536.45,Z 260.915,A -85,B 0,C 180,E1 26055.057,E2 26055.057} C_VEL
LIN {X 0,Y 536.463,Z 260.911,A -85,B 0,C 180,E1 26051.567,E2 26051.567} C_VEL
LIN {X 0,Y 536.448,Z 260.916,A -85,B 0,C 180,E1 26048.136,E2 26048.136} C_VEL
LIN {X 0,Y 536.51,Z 261.277,A -85,B 0,C 180,E1 26047.325,E2 26047.325} C_VEL
LIN {X 0,Y 544.186,Z 280.56,A -85,B 0,C 180,E1 26045.07,E2 26045.07} C_VEL
LIN {X 0,Y 544.545,Z 282.566,A -85,B 0,C 180,E1 26044.879,E2 26044.879} C_VEL
LIN {X 0,Y 542.884,Z 326.115,A -85,B 0,C 180,E1 26041.537,E2 26041.537} C_VEL
LIN {X 0,Y 542.962,Z 329.943,A -85,B 0,C 180,E1 26041.3,E2 26041.3} C_VEL
LIN {X 0,Y 544.949,Z 342.389,A -85,B 0,C 180,E1 26040.968,E2 26040.968} C_VEL
LIN {X 0,Y 542.963,Z 589.859,A -85,B 0,C 180,E1 26037.39,E2 26037.39} C_VEL
LIN {X 0,Y 542.504,Z 610.335,A -85,B 0,C 180,E1 26036.911,E2 26036.911} C_VEL
LIN {X 0,Y 541.955,Z 630.176,A -85,B 0,C 180,E1 26036.251,E2 26036.251} C_VEL
LIN {X 0,Y 541.263,Z 650.253,A -85,B 0,C 180,E1 26035.376,E2 26035.376} C_VEL
LIN {X 0,Y 540.529,Z 668.848,A -85,B 0,C 180,E1 26034.361,E2 26034.361} C_VEL
LIN {X 0,Y 539.755,Z 687.441,A -85,B 0,C 180,E1 26033.123,E2 26033.123} C_VEL
LIN {X 0,Y 538.948,Z 705.578,A -85,B 0,C 180,E1 26031.665,E2 26031.665} C_VEL
LIN {X 0,Y 538.199,Z 722.441,A -85,B 0,C 180,E1 26030.045,E2 26030.045} C_VEL
LIN {X 0,Y 537.547,Z 737.577,A -85,B 0,C 180,E1 26028.321,E2 26028.321} C_VEL
LIN {X 0,Y 537.018,Z 751.19,A -85,B 0,C 180,E1 26026.49,E2 26026.49} C_VEL
LIN {X 0,Y 536.602,Z 763.257,A -85,B 0,C 180,E1 26024.569,E2 26024.569} C_VEL
LIN {X 0,Y 536.299,Z 774.139,A -85,B 0,C 180,E1 26022.489,E2 26022.489} C_VEL
LIN {X 0,Y 536.097,Z 783.396,A -85,B 0,C 180,E1 26020.314,E2 26020.314} C_VEL
LIN {X 0,Y 535.999,Z 790.366,A -85,B 0,C 180,E1 26018.258,E2 26018.258} C_VEL
LIN {X 0,Y 535.941,Z 795.963,A -85,B 0,C 180,E1 26016.08,E2 26016.08} C_VEL
LIN {X 0,Y 535.919,Z 799.679,A -85,B 0,C 180,E1 26013.958,E2 26013.958} C_VEL
LIN {X 0,Y 535.911,Z 801.845,A -85,B 0,C 180,E1 26011.818,E2 26011.818} C_VEL
LIN {X 0,Y 535.904,Z 802.447,A -85,B 0,C 180,E1 26009.679,E2 26009.679} C_VEL
LIN {X 0,Y 535.904,Z 801.492,A -85,B 0,C 180,E1 26007.541,E2 26007.541} C_VEL
LIN {X 0,Y 535.916,Z 798.858,A -85,B 0,C 180,E1 26005.399,E2 26005.399} C_VEL
LIN {X 0,Y 535.946,Z 794.597,A -85,B 0,C 180,E1 26003.25,E2 26003.25} C_VEL
LIN {X 0,Y 536.008,Z 788.621,A -85,B 0,C 180,E1 26001.094,E2 26001.094} C_VEL
LIN {X 0,Y 536.133,Z 781.249,A -85,B 0,C 180,E1 25999.034,E2 25999.034} C_VEL
LIN {X 0,Y 536.349,Z 771.974,A -85,B 0,C 180,E1 25996.964,E2 25996.964} C_VEL
LIN {X 0,Y 536.669,Z 761.227,A -85,B 0,C 180,E1 25994.992,E2 25994.992} C_VEL
LIN {X 0,Y 537.091,Z 749.044,A -85,B 0,C 180,E1 25993.112,E2 25993.112} C_VEL
LIN {X 0,Y 537.62,Z 735.543,A -85,B 0,C 180,E1 25991.345,E2 25991.345} C_VEL
LIN {X 0,Y 538.271,Z 720.564,A -85,B 0,C 180,E1 25989.675,E2 25989.675} C_VEL
LIN {X 0,Y 538.987,Z 704.644,A -85,B 0,C 180,E1 25988.165,E2 25988.165} C_VEL
LIN {X 0,Y 539.781,Z 686.883,A -85,B 0,C 180,E1 25986.746,E2 25986.746} C_VEL
LIN {X 0,Y 540.56,Z 668.234,A -85,B 0,C 180,E1 25985.511,E2 25985.511} C_VEL
LIN {X 0,Y 541.281,Z 649.726,A -85,B 0,C 180,E1 25984.508,E2 25984.508} C_VEL
LIN {X 0,Y 541.97,Z 629.772,A -85,B 0,C 180,E1 25983.644,E2 25983.644} C_VEL
LIN {X 0,Y 542.525,Z 609.284,A -85,B 0,C 180,E1 25982.97,E2 25982.97} C_VEL
LIN {X 0,Y 542.971,Z 588.729,A -85,B 0,C 180,E1 25982.501,E2 25982.501} C_VEL
LIN {X 0,Y 544.933,Z 341.026,A -85,B 0,C 180,E1 25978.921,E2 25978.921} C_VEL
LIN {X 0,Y 542.819,Z 328.589,A -85,B 0,C 180,E1 25978.552,E2 25978.552} C_VEL
LIN {X 0,Y 544.448,Z 285.219,A -85,B 0,C 180,E1 25975.235,E2 25975.235} C_VEL
LIN {X 0,Y 544.421,Z 281.25,A -85,B 0,C 180,E1 25974.913,E2 25974.913} C_VEL
LIN {X 0,Y 537.553,Z 264.072,A -85,B 0,C 180,E1 25972.935,E2 25972.935} C_VEL
LIN {X 0,Y 536.485,Z 261.085,A -85,B 0,C 180,E1 25972.527,E2 25972.527} C_VEL
LIN {X 0,Y 536.464,Z 260.904,A -85,B 0,C 180,E1 25969.143,E2 25969.143} C_VEL
LIN {X 0,Y 536.448,Z 260.902,A -85,B 0,C 180,E1 25965.659,E2 25965.659} C_VEL
LIN {X 0,Y 536.461,Z 260.889,A -85,B 0,C 180,E1 25962.276,E2 25962.276} C_VEL
LIN {X 0,Y 536.447,Z 260.906,A -85,B 0,C 180,E1 25958.825,E2 25958.825} C_VEL
LIN {X 0,Y 536.458,Z 260.906,A -85,B 0,C 180,E1 25955.426,E2 25955.426} C_VEL
LIN {X 0,Y 536.462,Z 260.898,A -85,B 0,C 180,E1 25951.96,E2 25951.96} C_VEL
LIN {X 0,Y 536.437,Z 260.912,A -85,B 0,C 180,E1 25948.614,E2 25948.614} C_VEL
LIN {X 0,Y 536.461,Z 260.91,A -85,B 0,C 180,E1 25945.266,E2 25945.266} C_VEL
LIN {X 0,Y 536.462,Z 260.903,A -85,B 0,C 180,E1 25941.852,E2 25941.852} C_VEL
LIN {X 0,Y 536.426,Z 260.907,A -85,B 0,C 180,E1 25938.474,E2 25938.474} C_VEL
LIN {X 0,Y 536.452,Z 260.908,A -85,B 0,C 180,E1 25935.107,E2 25935.107} C_VEL
LIN {X 0,Y 536.459,Z 260.91,A -85,B 0,C 180,E1 25931.722,E2 25931.722} C_VEL
LIN {X 0,Y 536.414,Z 260.913,A -85,B 0,C 180,E1 25928.36,E2 25928.36} C_VEL
LIN {X 0,Y 536.442,Z 260.914,A -85,B 0,C 180,E1 25925.026,E2 25925.026} C_VEL
LIN {X 0,Y 536.442,Z 260.909,A -85,B 0,C 180,E1 25921.709,E2 25921.709} C_VEL
LIN {X 0,Y 536.401,Z 260.913,A -85,B 0,C 180,E1 25918.398,E2 25918.398} C_VEL
LIN {X 0,Y 536.442,Z 260.916,A -85,B 0,C 180,E1 25915.082,E2 25915.082} C_VEL
LIN {X 0,Y 536.407,Z 260.91,A -85,B 0,C 180,E1 25911.856,E2 25911.856} C_VEL
LIN {X 0,Y 536.389,Z 260.91,A -85,B 0,C 180,E1 25908.495,E2 25908.495} C_VEL
LIN {X 0,Y 536.453,Z 260.909,A -85,B 0,C 180,E1 25905.206,E2 25905.206} C_VEL
LIN {X 0,Y 536.391,Z 260.916,A -85,B 0,C 180,E1 25901.923,E2 25901.923} C_VEL
LIN {X 0,Y 536.394,Z 260.915,A -85,B 0,C 180,E1 25898.455,E2 25898.455} C_VEL
LIN {X 0,Y 536.457,Z 260.916,A -85,B 0,C 180,E1 25895.206,E2 25895.206} C_VEL
LIN {X 0,Y 536.399,Z 260.916,A -85,B 0,C 180,E1 25891.983,E2 25891.983} C_VEL
LIN {X 0,Y 536.422,Z 260.896,A -85,B 0,C 180,E1 25888.612,E2 25888.612} C_VEL
LIN {X 0,Y 536.451,Z 260.915,A -85,B 0,C 180,E1 25885.357,E2 25885.357} C_VEL
LIN {X 0,Y 536.411,Z 260.908,A -85,B 0,C 180,E1 25882.04,E2 25882.04} C_VEL
LIN {X 0,Y 536.45,Z 260.894,A -85,B 0,C 180,E1 25878.686,E2 25878.686} C_VEL
LIN {X 0,Y 536.451,Z 260.903,A -85,B 0,C 180,E1 25875.359,E2 25875.359} C_VEL
LIN {X 0,Y 536.423,Z 260.908,A -85,B 0,C 180,E1 25871.952,E2 25871.952} C_VEL
LIN {X 0,Y 536.471,Z 261.136,A -85,B 0,C 180,E1 25870.364,E2 25870.364} C_VEL
LIN {X 0,Y 537.892,Z 264.646,A -85,B 0,C 180,E1 25869.935,E2 25869.935} C_VEL
LIN {X 0,Y 546.447,Z 284.085,A -85,B 0,C 180,E1 25867.836,E2 25867.836} C_VEL
LIN {X 0,Y 545.928,Z 302.849,A -85,B 0,C 180,E1 25866.589,E2 25866.589} C_VEL
LIN {X 0,Y 548.125,Z 316.495,A -85,B 0,C 180,E1 25866.198,E2 25866.198} C_VEL
LIN {X 0,Y 546.051,Z 536.736,A -85,B 0,C 180,E1 25862.908,E2 25862.908} C_VEL
LIN {X 0,Y 545.343,Z 609.406,A -85,B 0,C 180,E1 25861.81,E2 25861.81} C_VEL
LIN {X 0,Y 544.74,Z 631.066,A -85,B 0,C 180,E1 25861.286,E2 25861.286} C_VEL
LIN {X 0,Y 544.046,Z 653.24,A -85,B 0,C 180,E1 25860.54,E2 25860.54} C_VEL
LIN {X 0,Y 543.251,Z 673.404,A -85,B 0,C 180,E1 25859.675,E2 25859.675} C_VEL
LIN {X 0,Y 542.322,Z 693.765,A -85,B 0,C 180,E1 25858.582,E2 25858.582} C_VEL
LIN {X 0,Y 541.316,Z 714.146,A -85,B 0,C 180,E1 25857.262,E2 25857.262} C_VEL
LIN {X 0,Y 540.362,Z 732.782,A -85,B 0,C 180,E1 25855.833,E2 25855.833} C_VEL
LIN {X 0,Y 539.449,Z 750.609,A -85,B 0,C 180,E1 25854.229,E2 25854.229} C_VEL
LIN {X 0,Y 538.587,Z 767.197,A -85,B 0,C 180,E1 25852.483,E2 25852.483} C_VEL
LIN {X 0,Y 537.832,Z 782.877,A -85,B 0,C 180,E1 25850.57,E2 25850.57} C_VEL
LIN {X 0,Y 537.225,Z 797.049,A -85,B 0,C 180,E1 25848.557,E2 25848.557} C_VEL
LIN {X 0,Y 536.747,Z 809.734,A -85,B 0,C 180,E1 25846.448,E2 25846.448} C_VEL
LIN {X 0,Y 536.402,Z 820.335,A -85,B 0,C 180,E1 25844.354,E2 25844.354} C_VEL
LIN {X 0,Y 536.157,Z 830.071,A -85,B 0,C 180,E1 25842.055,E2 25842.055} C_VEL
LIN {X 0,Y 536.021,Z 837.59,A -85,B 0,C 180,E1 25839.881,E2 25839.881} C_VEL
LIN {X 0,Y 535.949,Z 843.654,A -85,B 0,C 180,E1 25837.611,E2 25837.611} C_VEL
LIN {X 0,Y 535.923,Z 848.144,A -85,B 0,C 180,E1 25835.352,E2 25835.352} C_VEL
LIN {X 0,Y 535.916,Z 850.898,A -85,B 0,C 180,E1 25833.208,E2 25833.208} C_VEL
LIN {X 0,Y 535.907,Z 852.328,A -85,B 0,C 180,E1 25830.855,E2 25830.855} C_VEL
LIN {X 0,Y 535.901,Z 852.209,A -85,B 0,C 180,E1 25828.61,E2 25828.61} C_VEL
LIN {X 0,Y 535.906,Z 850.447,A -85,B 0,C 180,E1 25826.363,E2 25826.363} C_VEL
LIN {X 0,Y 535.925,Z 847.015,A -85,B 0,C 180,E1 25824.003,E2 25824.003} C_VEL
LIN {X 0,Y 535.972,Z 842.382,A -85,B 0,C 180,E1 25821.849,E2 25821.849} C_VEL
LIN {X 0,Y 536.055,Z 835.823,A -85,B 0,C 180,E1 25819.577,E2 25819.577} C_VEL
LIN {X 0,Y 536.212,Z 827.977,A -85,B 0,C 180,E1 25817.399,E2 25817.399} C_VEL
LIN {X 0,Y 536.464,Z 818.259,A -85,B 0,C 180,E1 25815.207,E2 25815.207} C_VEL
LIN {X 0,Y 536.853,Z 806.558,A -85,B 0,C 180,E1 25812.999,E2 25812.999} C_VEL
LIN {X 0,Y 537.381,Z 793.334,A -85,B 0,C 180,E1 25810.885,E2 25810.885} C_VEL
LIN {X 0,Y 538.047,Z 778.724,A -85,B 0,C 180,E1 25808.886,E2 25808.886} C_VEL
LIN {X 0,Y 538.795,Z 763.144,A -85,B 0,C 180,E1 25807.065,E2 25807.065} C_VEL
LIN {X 0,Y 539.645,Z 746.284,A -85,B 0,C 180,E1 25805.363,E2 25805.363} C_VEL
LIN {X 0,Y 540.625,Z 727.809,A -85,B 0,C 180,E1 25803.764,E2 25803.764} C_VEL
LIN {X 0,Y 541.579,Z 709.282,A -85,B 0,C 180,E1 25802.395,E2 25802.395} C_VEL
LIN {X 0,Y 542.497,Z 689.762,A -85,B 0,C 180,E1 25801.187,E2 25801.187} C_VEL
LIN {X 0,Y 543.45,Z 668.343,A -85,B 0,C 180,E1 25800.094,E2 25800.094} C_VEL
LIN {X 0,Y 544.265,Z 647.719,A -85,B 0,C 180,E1 25799.248,E2 25799.248} C_VEL
LIN {X 0,Y 544.893,Z 626.503,A -85,B 0,C 180,E1 25798.589,E2 25798.589} C_VEL
LIN {X 0,Y 545.404,Z 604.142,A -85,B 0,C 180,E1 25798.099,E2 25798.099} C_VEL
LIN {X 0,Y 547.512,Z 380.239,A -85,B 0,C 180,E1 25794.764,E2 25794.764} C_VEL
LIN {X 0,Y 547.945,Z 314.279,A -85,B 0,C 180,E1 25793.753,E2 25793.753} C_VEL
LIN {X 0,Y 545.841,Z 301.605,A -85,B 0,C 180,E1 25793.352,E2 25793.352} C_VEL
LIN {X 0,Y 546.419,Z 283.859,A -85,B 0,C 180,E1 25792.146,E2 25792.146} C_VEL
LIN {X 0,Y 537.636,Z 264.255,A -85,B 0,C 180,E1 25790.014,E2 25790.014} C_VEL
LIN {X 0,Y 536.471,Z 261.136,A -85,B 0,C 180,E1 25789.636,E2 25789.636} C_VEL
LIN {X 0,Y 536.434,Z 260.903,A -85,B 0,C 180,E1 25786.4,E2 25786.4} C_VEL
LIN {X 0,Y 536.466,Z 260.91,A -85,B 0,C 180,E1 25783.011,E2 25783.011} C_VEL
LIN {X 0,Y 536.418,Z 260.913,A -85,B 0,C 180,E1 25779.742,E2 25779.742} C_VEL
LIN {X 0,Y 536.425,Z 260.902,A -85,B 0,C 180,E1 25776.351,E2 25776.351} C_VEL
LIN {X 0,Y 536.462,Z 260.909,A -85,B 0,C 180,E1 25772.998,E2 25772.998} C_VEL
LIN {X 0,Y 536.404,Z 260.909,A -85,B 0,C 180,E1 25769.704,E2 25769.704} C_VEL
LIN {X 0,Y 536.414,Z 260.915,A -85,B 0,C 180,E1 25766.293,E2 25766.293} C_VEL
LIN {X 0,Y 536.442,Z 260.91,A -85,B 0,C 180,E1 25763.042,E2 25763.042} C_VEL
LIN {X 0,Y 536.388,Z 260.911,A -85,B 0,C 180,E1 25759.831,E2 25759.831} C_VEL
LIN {X 0,Y 536.436,Z 260.911,A -85,B 0,C 180,E1 25756.569,E2 25756.569} C_VEL
LIN {X 0,Y 536.393,Z 260.916,A -85,B 0,C 180,E1 25753.344,E2 25753.344} C_VEL
LIN {X 0,Y 536.392,Z 260.916,A -85,B 0,C 180,E1 25749.983,E2 25749.983} C_VEL
LIN {X 0,Y 536.458,Z 260.909,A -85,B 0,C 180,E1 25746.743,E2 25746.743} C_VEL
LIN {X 0,Y 536.398,Z 260.913,A -85,B 0,C 180,E1 25743.419,E2 25743.419} C_VEL
LIN {X 0,Y 536.411,Z 260.912,A -85,B 0,C 180,E1 25740,E2 25740} C_VEL
LIN {X 0,Y 536.452,Z 260.913,A -85,B 0,C 180,E1 25736.794,E2 25736.794} C_VEL
LIN {X 0,Y 536.407,Z 260.909,A -85,B 0,C 180,E1 25733.453,E2 25733.453} C_VEL
LIN {X 0,Y 536.44,Z 260.904,A -85,B 0,C 180,E1 25730.126,E2 25730.126} C_VEL
LIN {X 0,Y 536.448,Z 260.916,A -85,B 0,C 180,E1 25726.856,E2 25726.856} C_VEL
LIN {X 0,Y 536.421,Z 260.912,A -85,B 0,C 180,E1 25723.541,E2 25723.541} C_VEL
LIN {X 0,Y 536.46,Z 260.909,A -85,B 0,C 180,E1 25720.171,E2 25720.171} C_VEL
LIN {X 0,Y 536.46,Z 260.91,A -85,B 0,C 180,E1 25716.726,E2 25716.726} C_VEL
LIN {X 0,Y 536.432,Z 260.907,A -85,B 0,C 180,E1 25713.307,E2 25713.307} C_VEL
LIN {X 0,Y 536.458,Z 260.897,A -85,B 0,C 180,E1 25709.909,E2 25709.909} C_VEL
LIN {X 0,Y 536.461,Z 260.912,A -85,B 0,C 180,E1 25706.517,E2 25706.517} C_VEL
LIN {X 0,Y 536.44,Z 260.912,A -85,B 0,C 180,E1 25705.355,E2 25705.355} C_VEL
LIN {X 0,Y 535.452,Z 261.038,A -85,B 0,C 180,E1 25704.532,E2 25704.532} C_VEL
LIN {X 0,Y 528.966,Z 261.834,A -85,B 0,C 180,E1 25702.161,E2 25702.161} C_VEL
LIN {X 0,Y 528.512,Z 261.891,A -85,B 0,C 180,E1 25701.618,E2 25701.618} C_VEL
LIN {X 0,Y 528.514,Z 261.881,A -85,B 0,C 180,E1 25698.19,E2 25698.19} C_VEL
LIN {X 0,Y 528.521,Z 261.896,A -85,B 0,C 180,E1 25694.727,E2 25694.727} C_VEL
LIN {X 0,Y 528.515,Z 261.903,A -85,B 0,C 180,E1 25691.317,E2 25691.317} C_VEL
LIN {X 0,Y 528.534,Z 262.069,A -85,B 0,C 180,E1 25688.006,E2 25688.006} C_VEL
LIN {X 0,Y 528.907,Z 263.553,A -85,B 0,C 180,E1 25687.769,E2 25687.769} C_VEL
LIN {X 0,Y 535.996,Z 280.578,A -85,B 0,C 180,E1 25685.722,E2 25685.722} C_VEL
LIN {X 0,Y 537.637,Z 285.231,A -85,B 0,C 180,E1 25685.205,E2 25685.205} C_VEL
LIN {X 0,Y 535.849,Z 328.228,A -85,B 0,C 180,E1 25681.873,E2 25681.873} C_VEL
LIN {X 0,Y 538.283,Z 343.704,A -85,B 0,C 180,E1 25681.422,E2 25681.422} C_VEL
LIN {X 0,Y 536.074,Z 570.407,A -85,B 0,C 180,E1 25678.089,E2 25678.089} C_VEL
LIN {X 0,Y 535.688,Z 596.639,A -85,B 0,C 180,E1 25677.645,E2 25677.645} C_VEL
LIN {X 0,Y 535.154,Z 617.591,A -85,B 0,C 180,E1 25677.079,E2 25677.079} C_VEL
LIN {X 0,Y 534.502,Z 637.073,A -85,B 0,C 180,E1 25676.358,E2 25676.358} C_VEL
LIN {X 0,Y 533.733,Z 656.106,A -85,B 0,C 180,E1 25675.452,E2 25675.452} C_VEL
LIN {X 0,Y 532.903,Z 674.257,A -85,B 0,C 180,E1 25674.379,E2 25674.379} C_VEL
LIN {X 0,Y 532.032,Z 691.857,A -85,B 0,C 180,E1 25673.127,E2 25673.127} C_VEL
LIN {X 0,Y 531.156,Z 709.25,A -85,B 0,C 180,E1 25671.65,E2 25671.65} C_VEL
LIN {X 0,Y 530.38,Z 725.028,A -85,B 0,C 180,E1 25670.065,E2 25670.065} C_VEL
LIN {X 0,Y 529.703,Z 739.379,A -85,B 0,C 180,E1 25668.374,E2 25668.374} C_VEL
LIN {X 0,Y 529.109,Z 753.082,A -85,B 0,C 180,E1 25666.466,E2 25666.466} C_VEL
LIN {X 0,Y 528.643,Z 765.231,A -85,B 0,C 180,E1 25664.446,E2 25664.446} C_VEL
LIN {X 0,Y 528.327,Z 775.272,A -85,B 0,C 180,E1 25662.437,E2 25662.437} C_VEL
LIN {X 0,Y 528.117,Z 783.804,A -85,B 0,C 180,E1 25660.361,E2 25660.361} C_VEL
LIN {X 0,Y 527.998,Z 790.974,A -85,B 0,C 180,E1 25658.165,E2 25658.165} C_VEL
LIN {X 0,Y 527.941,Z 796.349,A -85,B 0,C 180,E1 25655.979,E2 25655.979} C_VEL
LIN {X 0,Y 527.917,Z 799.997,A -85,B 0,C 180,E1 25653.801,E2 25653.801} C_VEL
LIN {X 0,Y 527.904,Z 801.979,A -85,B 0,C 180,E1 25651.628,E2 25651.628} C_VEL
LIN {X 0,Y 527.901,Z 802.38,A -85,B 0,C 180,E1 25649.349,E2 25649.349} C_VEL
LIN {X 0,Y 527.911,Z 801.054,A -85,B 0,C 180,E1 25647.069,E2 25647.069} C_VEL
LIN {X 0,Y 527.924,Z 798.167,A -85,B 0,C 180,E1 25644.893,E2 25644.893} C_VEL
LIN {X 0,Y 527.962,Z 793.578,A -85,B 0,C 180,E1 25642.711,E2 25642.711} C_VEL
LIN {X 0,Y 528.051,Z 787.398,A -85,B 0,C 180,E1 25640.579,E2 25640.579} C_VEL
LIN {X 0,Y 528.217,Z 779.407,A -85,B 0,C 180,E1 25638.426,E2 25638.426} C_VEL
LIN {X 0,Y 528.491,Z 769.723,A -85,B 0,C 180,E1 25636.321,E2 25636.321} C_VEL
LIN {X 0,Y 528.859,Z 759.273,A -85,B 0,C 180,E1 25634.428,E2 25634.428} C_VEL
LIN {X 0,Y 529.376,Z 746.726,A -85,B 0,C 180,E1 25632.52,E2 25632.52} C_VEL
LIN {X 0,Y 530.006,Z 732.751,A -85,B 0,C 180,E1 25630.723,E2 25630.723} C_VEL
LIN {X 0,Y 530.731,Z 717.775,A -85,B 0,C 180,E1 25629.084,E2 25629.084} C_VEL
LIN {X 0,Y 531.59,Z 700.638,A -85,B 0,C 180,E1 25627.496,E2 25627.496} C_VEL
LIN {X 0,Y 532.508,Z 682.267,A -85,B 0,C 180,E1 25626.074,E2 25626.074} C_VEL
LIN {X 0,Y 533.402,Z 663.534,A -85,B 0,C 180,E1 25624.875,E2 25624.875} C_VEL
LIN {X 0,Y 534.186,Z 645.047,A -85,B 0,C 180,E1 25623.906,E2 25623.906} C_VEL
LIN {X 0,Y 534.934,Z 624.862,A -85,B 0,C 180,E1 25623.072,E2 25623.072} C_VEL
LIN {X 0,Y 535.539,Z 604.508,A -85,B 0,C 180,E1 25622.451,E2 25622.451} C_VEL
LIN {X 0,Y 535.922,Z 584.077,A -85,B 0,C 180,E1 25622.027,E2 25622.027} C_VEL
LIN {X 0,Y 538.281,Z 344.377,A -85,B 0,C 180,E1 25618.497,E2 25618.497} C_VEL
LIN {X 0,Y 537.753,Z 339.485,A -85,B 0,C 180,E1 25618.383,E2 25618.383} C_VEL
LIN {X 0,Y 535.84,Z 328.357,A -85,B 0,C 180,E1 25618.047,E2 25618.047} C_VEL
LIN {X 0,Y 537.645,Z 285.156,A -85,B 0,C 180,E1 25614.698,E2 25614.698} C_VEL
LIN {X 0,Y 531.448,Z 269.215,A -85,B 0,C 180,E1 25612.85,E2 25612.85} C_VEL
LIN {X 0,Y 528.548,Z 262.195,A -85,B 0,C 180,E1 25611.953,E2 25611.953} C_VEL
LIN {X 0,Y 528.504,Z 261.883,A -85,B 0,C 180,E1 25609.846,E2 25609.846} C_VEL
LIN {X 0,Y 528.52,Z 261.883,A -85,B 0,C 180,E1 25606.433,E2 25606.433} C_VEL
LIN {X 0,Y 528.513,Z 261.882,A -85,B 0,C 180,E1 25602.927,E2 25602.927} C_VEL
LIN {X 0,Y 528.519,Z 261.903,A -85,B 0,C 180,E1 25599.468,E2 25599.468} C_VEL
LIN {X 0,Y 528.522,Z 261.888,A -85,B 0,C 180,E1 25595.936,E2 25595.936} C_VEL
LIN {X 0,Y 528.502,Z 261.889,A -85,B 0,C 180,E1 25592.5,E2 25592.5} C_VEL
LIN {X 0,Y 528.519,Z 261.898,A -85,B 0,C 180,E1 25589.074,E2 25589.074} C_VEL
LIN {X 0,Y 528.523,Z 261.893,A -85,B 0,C 180,E1 25585.672,E2 25585.672} C_VEL
LIN {X 0,Y 528.5,Z 261.893,A -85,B 0,C 180,E1 25582.233,E2 25582.233} C_VEL
LIN {X 0,Y 528.492,Z 261.897,A -85,B 0,C 180,E1 25578.761,E2 25578.761} C_VEL
LIN {X 0,Y 528.529,Z 261.899,A -85,B 0,C 180,E1 25575.358,E2 25575.358} C_VEL
LIN {X 0,Y 528.496,Z 261.9,A -85,B 0,C 180,E1 25572.012,E2 25572.012} C_VEL
LIN {X 0,Y 528.478,Z 261.903,A -85,B 0,C 180,E1 25568.596,E2 25568.596} C_VEL
LIN {X 0,Y 528.525,Z 261.895,A -85,B 0,C 180,E1 25565.319,E2 25565.319} C_VEL
LIN {X 0,Y 528.482,Z 261.898,A -85,B 0,C 180,E1 25561.952,E2 25561.952} C_VEL
LIN {X 0,Y 528.467,Z 261.902,A -85,B 0,C 180,E1 25558.591,E2 25558.591} C_VEL
LIN {X 0,Y 528.521,Z 261.901,A -85,B 0,C 180,E1 25555.334,E2 25555.334} C_VEL
LIN {X 0,Y 528.457,Z 261.899,A -85,B 0,C 180,E1 25552.061,E2 25552.061} C_VEL
LIN {X 0,Y 528.453,Z 261.899,A -85,B 0,C 180,E1 25548.537,E2 25548.537} C_VEL
LIN {X 0,Y 528.511,Z 261.9,A -85,B 0,C 180,E1 25545.315,E2 25545.315} C_VEL
LIN {X 0,Y 528.447,Z 261.905,A -85,B 0,C 180,E1 25542.037,E2 25542.037} C_VEL
LIN {X 0,Y 528.46,Z 261.904,A -85,B 0,C 180,E1 25538.567,E2 25538.567} C_VEL
LIN {X 0,Y 528.501,Z 261.903,A -85,B 0,C 180,E1 25535.405,E2 25535.405} C_VEL
LIN {X 0,Y 528.459,Z 261.905,A -85,B 0,C 180,E1 25532.074,E2 25532.074} C_VEL
LIN {X 0,Y 528.498,Z 261.881,A -85,B 0,C 180,E1 25528.772,E2 25528.772} C_VEL
LIN {X 0,Y 528.505,Z 261.906,A -85,B 0,C 180,E1 25525.42,E2 25525.42} C_VEL
LIN {X 0,Y 528.472,Z 261.896,A -85,B 0,C 180,E1 25522.056,E2 25522.056} C_VEL
LIN {X 0,Y 528.51,Z 261.882,A -85,B 0,C 180,E1 25518.681,E2 25518.681} C_VEL
LIN {X 0,Y 528.518,Z 261.888,A -85,B 0,C 180,E1 25515.271,E2 25515.271} C_VEL
LIN {X 0,Y 528.485,Z 261.893,A -85,B 0,C 180,E1 25511.9,E2 25511.9} C_VEL
LIN {X 0,Y 528.572,Z 262.204,A -85,B 0,C 180,E1 25510.959,E2 25510.959} C_VEL
LIN {X 0,Y 533.124,Z 272.761,A -85,B 0,C 180,E1 25509.741,E2 25509.741} C_VEL
LIN {X 0,Y 539.677,Z 287.557,A -85,B 0,C 180,E1 25508.143,E2 25508.143} C_VEL
LIN {X 0,Y 539.205,Z 302.782,A -85,B 0,C 180,E1 25507.122,E2 25507.122} C_VEL
LIN {X 0,Y 541.654,Z 317.962,A -85,B 0,C 180,E1 25506.677,E2 25506.677} C_VEL
LIN {X 0,Y 539.327,Z 537.754,A -85,B 0,C 180,E1 25503.356,E2 25503.356} C_VEL
LIN {X 0,Y 538.542,Z 609.405,A -85,B 0,C 180,E1 25502.26,E2 25502.26} C_VEL
LIN {X 0,Y 537.875,Z 631.064,A -85,B 0,C 180,E1 25501.731,E2 25501.731} C_VEL
LIN {X 0,Y 537.103,Z 653.236,A -85,B 0,C 180,E1 25500.978,E2 25500.978} C_VEL
LIN {X 0,Y 536.193,Z 673.686,A -85,B 0,C 180,E1 25500.091,E2 25500.091} C_VEL
LIN {X 0,Y 535.177,Z 693.668,A -85,B 0,C 180,E1 25499.006,E2 25499.006} C_VEL
LIN {X 0,Y 534.037,Z 714.142,A -85,B 0,C 180,E1 25497.665,E2 25497.665} C_VEL
LIN {X 0,Y 532.979,Z 732.779,A -85,B 0,C 180,E1 25496.218,E2 25496.218} C_VEL
LIN {X 0,Y 531.947,Z 750.517,A -85,B 0,C 180,E1 25494.603,E2 25494.603} C_VEL
LIN {X 0,Y 530.99,Z 766.69,A -85,B 0,C 180,E1 25492.882,E2 25492.882} C_VEL
LIN {X 0,Y 530.11,Z 782.877,A -85,B 0,C 180,E1 25490.884,E2 25490.884} C_VEL
LIN {X 0,Y 529.419,Z 797.051,A -85,B 0,C 180,E1 25488.841,E2 25488.841} C_VEL
LIN {X 0,Y 528.877,Z 809.732,A -85,B 0,C 180,E1 25486.7,E2 25486.7} C_VEL
LIN {X 0,Y 528.483,Z 820.334,A -85,B 0,C 180,E1 25484.573,E2 25484.573} C_VEL
LIN {X 0,Y 528.198,Z 830.072,A -85,B 0,C 180,E1 25482.24,E2 25482.24} C_VEL
LIN {X 0,Y 528.043,Z 837.59,A -85,B 0,C 180,E1 25480.032,E2 25480.032} C_VEL
LIN {X 0,Y 527.958,Z 843.654,A -85,B 0,C 180,E1 25477.727,E2 25477.727} C_VEL
LIN {X 0,Y 527.926,Z 848.144,A -85,B 0,C 180,E1 25475.434,E2 25475.434} C_VEL
LIN {X 0,Y 527.916,Z 850.898,A -85,B 0,C 180,E1 25473.257,E2 25473.257} C_VEL
LIN {X 0,Y 527.908,Z 852.328,A -85,B 0,C 180,E1 25470.868,E2 25470.868} C_VEL
LIN {X 0,Y 527.9,Z 852.209,A -85,B 0,C 180,E1 25468.589,E2 25468.589} C_VEL
LIN {X 0,Y 527.905,Z 850.447,A -85,B 0,C 180,E1 25466.308,E2 25466.308} C_VEL
LIN {X 0,Y 527.929,Z 846.961,A -85,B 0,C 180,E1 25463.883,E2 25463.883} C_VEL
LIN {X 0,Y 527.98,Z 842.383,A -85,B 0,C 180,E1 25461.725,E2 25461.725} C_VEL
LIN {X 0,Y 528.073,Z 835.823,A -85,B 0,C 180,E1 25459.417,E2 25459.417} C_VEL
LIN {X 0,Y 528.255,Z 827.976,A -85,B 0,C 180,E1 25457.206,E2 25457.206} C_VEL
LIN {X 0,Y 528.545,Z 818.26,A -85,B 0,C 180,E1 25454.98,E2 25454.98} C_VEL
LIN {X 0,Y 528.967,Z 807.193,A -85,B 0,C 180,E1 25452.851,E2 25452.851} C_VEL
LIN {X 0,Y 529.552,Z 794.36,A -85,B 0,C 180,E1 25450.744,E2 25450.744} C_VEL
LIN {X 0,Y 530.321,Z 779.391,A -85,B 0,C 180,E1 25448.65,E2 25448.65} C_VEL
LIN {X 0,Y 531.175,Z 763.65,A -85,B 0,C 180,E1 25446.775,E2 25446.775} C_VEL
LIN {X 0,Y 532.163,Z 746.282,A -85,B 0,C 180,E1 25444.993,E2 25444.993} C_VEL
LIN {X 0,Y 533.263,Z 727.864,A -85,B 0,C 180,E1 25443.378,E2 25443.378} C_VEL
LIN {X 0,Y 534.347,Z 709.279,A -85,B 0,C 180,E1 25441.988,E2 25441.988} C_VEL
LIN {X 0,Y 535.365,Z 689.759,A -85,B 0,C 180,E1 25440.767,E2 25440.767} C_VEL
LIN {X 0,Y 536.449,Z 668.081,A -85,B 0,C 180,E1 25439.65,E2 25439.65} C_VEL
LIN {X 0,Y 537.339,Z 647.506,A -85,B 0,C 180,E1 25438.8,E2 25438.8} C_VEL
LIN {X 0,Y 538.052,Z 626.391,A -85,B 0,C 180,E1 25438.139,E2 25438.139} C_VEL
LIN {X 0,Y 538.611,Z 603.93,A -85,B 0,C 180,E1 25437.644,E2 25437.644} C_VEL
LIN {X 0,Y 540.967,Z 381.511,A -85,B 0,C 180,E1 25434.293,E2 25434.293} C_VEL
LIN {X 0,Y 541.483,Z 315.782,A -85,B 0,C 180,E1 25433.274,E2 25433.274} C_VEL
LIN {X 0,Y 539.127,Z 301.834,A -85,B 0,C 180,E1 25432.835,E2 25432.835} C_VEL
LIN {X 0,Y 539.6,Z 287.182,A -85,B 0,C 180,E1 25431.824,E2 25431.824} C_VEL
LIN {X 0,Y 528.599,Z 262.353,A -85,B 0,C 180,E1 25429.07,E2 25429.07} C_VEL
LIN {X 0,Y 528.517,Z 261.88,A -85,B 0,C 180,E1 25428.681,E2 25428.681} C_VEL
LIN {X 0,Y 528.518,Z 261.881,A -85,B 0,C 180,E1 25425.273,E2 25425.273} C_VEL
LIN {X 0,Y 528.477,Z 261.886,A -85,B 0,C 180,E1 25421.902,E2 25421.902} C_VEL
LIN {X 0,Y 528.498,Z 261.898,A -85,B 0,C 180,E1 25418.494,E2 25418.494} C_VEL
LIN {X 0,Y 528.519,Z 261.894,A -85,B 0,C 180,E1 25415.107,E2 25415.107} C_VEL
LIN {X 0,Y 528.465,Z 261.888,A -85,B 0,C 180,E1 25411.844,E2 25411.844} C_VEL
LIN {X 0,Y 528.494,Z 261.905,A -85,B 0,C 180,E1 25408.474,E2 25408.474} C_VEL
LIN {X 0,Y 528.49,Z 261.902,A -85,B 0,C 180,E1 25405.194,E2 25405.194} C_VEL
LIN {X 0,Y 528.455,Z 261.904,A -85,B 0,C 180,E1 25401.884,E2 25401.884} C_VEL
LIN {X 0,Y 528.503,Z 261.902,A -85,B 0,C 180,E1 25398.594,E2 25398.594} C_VEL
LIN {X 0,Y 528.455,Z 261.899,A -85,B 0,C 180,E1 25395.36,E2 25395.36} C_VEL
LIN {X 0,Y 528.445,Z 261.899,A -85,B 0,C 180,E1 25391.902,E2 25391.902} C_VEL
LIN {X 0,Y 528.512,Z 261.9,A -85,B 0,C 180,E1 25388.595,E2 25388.595} C_VEL
LIN {X 0,Y 528.462,Z 261.904,A -85,B 0,C 180,E1 25385.319,E2 25385.319} C_VEL
LIN {X 0,Y 528.461,Z 261.902,A -85,B 0,C 180,E1 25381.843,E2 25381.843} C_VEL
LIN {X 0,Y 528.525,Z 261.895,A -85,B 0,C 180,E1 25378.591,E2 25378.591} C_VEL
LIN {X 0,Y 528.476,Z 261.904,A -85,B 0,C 180,E1 25375.225,E2 25375.225} C_VEL
LIN {X 0,Y 528.475,Z 261.902,A -85,B 0,C 180,E1 25371.733,E2 25371.733} C_VEL
LIN {X 0,Y 528.527,Z 261.901,A -85,B 0,C 180,E1 25368.432,E2 25368.432} C_VEL
LIN {X 0,Y 528.493,Z 261.897,A -85,B 0,C 180,E1 25365.09,E2 25365.09} C_VEL
LIN {X 0,Y 528.488,Z 261.895,A -85,B 0,C 180,E1 25361.696,E2 25361.696} C_VEL
LIN {X 0,Y 528.527,Z 261.894,A -85,B 0,C 180,E1 25358.352,E2 25358.352} C_VEL
LIN {X 0,Y 528.508,Z 261.904,A -85,B 0,C 180,E1 25354.927,E2 25354.927} C_VEL
LIN {X 0,Y 528.496,Z 261.9,A -85,B 0,C 180,E1 25351.526,E2 25351.526} C_VEL
LIN {X 0,Y 528.522,Z 261.882,A -85,B 0,C 180,E1 25348.142,E2 25348.142} C_VEL
LIN {X 0,Y 528.522,Z 261.896,A -85,B 0,C 180,E1 25344.627,E2 25344.627} C_VEL
LIN {X 0,Y 528.512,Z 261.891,A -85,B 0,C 180,E1 25341.618,E2 25341.618} C_VEL
LIN {X 0,Y 527.503,Z 262.026,A -85,B 0,C 180,E1 25340.784,E2 25340.784} C_VEL
LIN {X 0,Y 521.021,Z 262.816,A -85,B 0,C 180,E1 25338.377,E2 25338.377} C_VEL
LIN {X 0,Y 520.582,Z 262.865,A -85,B 0,C 180,E1 25337.826,E2 25337.826} C_VEL
LIN {X 0,Y 520.576,Z 262.879,A -85,B 0,C 180,E1 25334.355,E2 25334.355} C_VEL
LIN {X 0,Y 520.583,Z 262.882,A -85,B 0,C 180,E1 25330.822,E2 25330.822} C_VEL
LIN {X 0,Y 520.614,Z 263.108,A -85,B 0,C 180,E1 25328.606,E2 25328.606} C_VEL
LIN {X 0,Y 523.098,Z 269.389,A -85,B 0,C 180,E1 25327.779,E2 25327.779} C_VEL
LIN {X 0,Y 530.493,Z 287.639,A -85,B 0,C 180,E1 25325.582,E2 25325.582} C_VEL
LIN {X 0,Y 530.614,Z 290.64,A -85,B 0,C 180,E1 25325.321,E2 25325.321} C_VEL
LIN {X 0,Y 528.96,Z 328.828,A -85,B 0,C 180,E1 25322.347,E2 25322.347} C_VEL
LIN {X 0,Y 531.654,Z 345.066,A -85,B 0,C 180,E1 25321.887,E2 25321.887} C_VEL
LIN {X 0,Y 528.959,Z 581.502,A -85,B 0,C 180,E1 25318.344,E2 25318.344} C_VEL
LIN {X 0,Y 528.503,Z 602.409,A -85,B 0,C 180,E1 25317.918,E2 25317.918} C_VEL
LIN {X 0,Y 527.805,Z 623.206,A -85,B 0,C 180,E1 25317.291,E2 25317.291} C_VEL
LIN {X 0,Y 527.075,Z 641.831,A -85,B 0,C 180,E1 25316.534,E2 25316.534} C_VEL
LIN {X 0,Y 526.174,Z 661.042,A -85,B 0,C 180,E1 25315.553,E2 25315.553} C_VEL
LIN {X 0,Y 525.24,Z 679.408,A -85,B 0,C 180,E1 25314.398,E2 25314.398} C_VEL
LIN {X 0,Y 524.291,Z 696.941,A -85,B 0,C 180,E1 25313.072,E2 25313.072} C_VEL
LIN {X 0,Y 523.316,Z 714.109,A -85,B 0,C 180,E1 25311.52,E2 25311.52} C_VEL
LIN {X 0,Y 522.43,Z 730.098,A -85,B 0,C 180,E1 25309.8,E2 25309.8} C_VEL
LIN {X 0,Y 521.67,Z 744.46,A -85,B 0,C 180,E1 25307.973,E2 25307.973} C_VEL
LIN {X 0,Y 521.07,Z 757.312,A -85,B 0,C 180,E1 25306.04,E2 25306.04} C_VEL
LIN {X 0,Y 520.605,Z 768.689,A -85,B 0,C 180,E1 25304.004,E2 25304.004} C_VEL
LIN {X 0,Y 520.275,Z 778.578,A -85,B 0,C 180,E1 25301.866,E2 25301.866} C_VEL
LIN {X 0,Y 520.085,Z 786.564,A -85,B 0,C 180,E1 25299.74,E2 25299.74} C_VEL
LIN {X 0,Y 519.973,Z 793.096,A -85,B 0,C 180,E1 25297.513,E2 25297.513} C_VEL
LIN {X 0,Y 519.922,Z 797.796,A -85,B 0,C 180,E1 25295.296,E2 25295.296} C_VEL
LIN {X 0,Y 519.911,Z 800.848,A -85,B 0,C 180,E1 25293.087,E2 25293.087} C_VEL
LIN {X 0,Y 519.91,Z 802.338,A -85,B 0,C 180,E1 25290.771,E2 25290.771} C_VEL
LIN {X 0,Y 519.901,Z 802.169,A -85,B 0,C 180,E1 25288.567,E2 25288.567} C_VEL
LIN {X 0,Y 519.908,Z 800.373,A -85,B 0,C 180,E1 25286.361,E2 25286.361} C_VEL
LIN {X 0,Y 519.936,Z 796.932,A -85,B 0,C 180,E1 25284.15,E2 25284.15} C_VEL
LIN {X 0,Y 519.997,Z 791.828,A -85,B 0,C 180,E1 25281.931,E2 25281.931} C_VEL
LIN {X 0,Y 520.111,Z 785.35,A -85,B 0,C 180,E1 25279.813,E2 25279.813} C_VEL
LIN {X 0,Y 520.327,Z 777.1,A -85,B 0,C 180,E1 25277.685,E2 25277.685} C_VEL
LIN {X 0,Y 520.681,Z 766.843,A -85,B 0,C 180,E1 25275.544,E2 25275.544} C_VEL
LIN {X 0,Y 521.143,Z 755.623,A -85,B 0,C 180,E1 25273.597,E2 25273.597} C_VEL
LIN {X 0,Y 521.761,Z 742.581,A -85,B 0,C 180,E1 25271.683,E2 25271.683} C_VEL
LIN {X 0,Y 522.537,Z 727.846,A -85,B 0,C 180,E1 25269.854,E2 25269.854} C_VEL
LIN {X 0,Y 523.391,Z 712.627,A -85,B 0,C 180,E1 25268.248,E2 25268.248} C_VEL
LIN {X 0,Y 524.348,Z 695.91,A -85,B 0,C 180,E1 25266.752,E2 25266.752} C_VEL
LIN {X 0,Y 525.365,Z 677.37,A -85,B 0,C 180,E1 25265.368,E2 25265.368} C_VEL
LIN {X 0,Y 526.306,Z 658.51,A -85,B 0,C 180,E1 25264.213,E2 25264.213} C_VEL
LIN {X 0,Y 527.158,Z 639.88,A -85,B 0,C 180,E1 25263.288,E2 25263.288} C_VEL
LIN {X 0,Y 527.944,Z 619.3,A -85,B 0,C 180,E1 25262.489,E2 25262.489} C_VEL
LIN {X 0,Y 528.573,Z 598.57,A -85,B 0,C 180,E1 25261.901,E2 25261.901} C_VEL
LIN {X 0,Y 529.026,Z 576.732,A -85,B 0,C 180,E1 25261.492,E2 25261.492} C_VEL
LIN {X 0,Y 531.658,Z 343.938,A -85,B 0,C 180,E1 25258.006,E2 25258.006} C_VEL
LIN {X 0,Y 528.902,Z 328.124,A -85,B 0,C 180,E1 25257.529,E2 25257.529} C_VEL
LIN {X 0,Y 530.729,Z 288.274,A -85,B 0,C 180,E1 25254.4,E2 25254.4} C_VEL
LIN {X 0,Y 523.554,Z 270.238,A -85,B 0,C 180,E1 25252.245,E2 25252.245} C_VEL
LIN {X 0,Y 520.649,Z 263.33,A -85,B 0,C 180,E1 25251.353,E2 25251.353} C_VEL
LIN {X 0,Y 520.575,Z 262.871,A -85,B 0,C 180,E1 25250.811,E2 25250.811} C_VEL
LIN {X 0,Y 520.577,Z 262.875,A -85,B 0,C 180,E1 25247.36,E2 25247.36} C_VEL
LIN {X 0,Y 520.577,Z 262.89,A -85,B 0,C 180,E1 25243.897,E2 25243.897} C_VEL
LIN {X 0,Y 520.576,Z 262.888,A -85,B 0,C 180,E1 25240.481,E2 25240.481} C_VEL
LIN {X 0,Y 520.571,Z 262.87,A -85,B 0,C 180,E1 25236.955,E2 25236.955} C_VEL
LIN {X 0,Y 520.582,Z 262.889,A -85,B 0,C 180,E1 25233.452,E2 25233.452} C_VEL
LIN {X 0,Y 520.59,Z 262.872,A -85,B 0,C 180,E1 25229.958,E2 25229.958} C_VEL
LIN {X 0,Y 520.559,Z 262.883,A -85,B 0,C 180,E1 25226.487,E2 25226.487} C_VEL
LIN {X 0,Y 520.575,Z 262.885,A -85,B 0,C 180,E1 25223.068,E2 25223.068} C_VEL
LIN {X 0,Y 520.589,Z 262.888,A -85,B 0,C 180,E1 25219.64,E2 25219.64} C_VEL
LIN {X 0,Y 520.549,Z 262.889,A -85,B 0,C 180,E1 25216.286,E2 25216.286} C_VEL
LIN {X 0,Y 520.549,Z 262.892,A -85,B 0,C 180,E1 25212.761,E2 25212.761} C_VEL
LIN {X 0,Y 520.588,Z 262.882,A -85,B 0,C 180,E1 25209.396,E2 25209.396} C_VEL
LIN {X 0,Y 520.544,Z 262.883,A -85,B 0,C 180,E1 25206.064,E2 25206.064} C_VEL
LIN {X 0,Y 520.535,Z 262.889,A -85,B 0,C 180,E1 25202.642,E2 25202.642} C_VEL
LIN {X 0,Y 520.59,Z 262.891,A -85,B 0,C 180,E1 25199.34,E2 25199.34} C_VEL
LIN {X 0,Y 520.527,Z 262.889,A -85,B 0,C 180,E1 25196.035,E2 25196.035} C_VEL
LIN {X 0,Y 520.521,Z 262.889,A -85,B 0,C 180,E1 25192.606,E2 25192.606} C_VEL
LIN {X 0,Y 520.573,Z 262.887,A -85,B 0,C 180,E1 25189.263,E2 25189.263} C_VEL
LIN {X 0,Y 520.513,Z 262.894,A -85,B 0,C 180,E1 25185.938,E2 25185.938} C_VEL
LIN {X 0,Y 520.508,Z 262.894,A -85,B 0,C 180,E1 25182.447,E2 25182.447} C_VEL
LIN {X 0,Y 520.578,Z 262.891,A -85,B 0,C 180,E1 25179.187,E2 25179.187} C_VEL
LIN {X 0,Y 520.525,Z 262.892,A -85,B 0,C 180,E1 25175.837,E2 25175.837} C_VEL
LIN {X 0,Y 520.525,Z 262.893,A -85,B 0,C 180,E1 25172.312,E2 25172.312} C_VEL
LIN {X 0,Y 520.583,Z 262.866,A -85,B 0,C 180,E1 25169.021,E2 25169.021} C_VEL
LIN {X 0,Y 520.548,Z 262.895,A -85,B 0,C 180,E1 25165.618,E2 25165.618} C_VEL
LIN {X 0,Y 520.535,Z 262.884,A -85,B 0,C 180,E1 25162.133,E2 25162.133} C_VEL
LIN {X 0,Y 520.581,Z 262.868,A -85,B 0,C 180,E1 25158.793,E2 25158.793} C_VEL
LIN {X 0,Y 520.575,Z 262.876,A -85,B 0,C 180,E1 25155.335,E2 25155.335} C_VEL
LIN {X 0,Y 520.546,Z 262.88,A -85,B 0,C 180,E1 25151.945,E2 25151.945} C_VEL
LIN {X 0,Y 520.64,Z 263.391,A -85,B 0,C 180,E1 25151.57,E2 25151.57} C_VEL
LIN {X 0,Y 532.66,Z 290.517,A -85,B 0,C 180,E1 25148.487,E2 25148.487} C_VEL
LIN {X 0,Y 532.504,Z 302.985,A -85,B 0,C 180,E1 25147.647,E2 25147.647} C_VEL
LIN {X 0,Y 535.222,Z 319.472,A -85,B 0,C 180,E1 25147.166,E2 25147.166} C_VEL
LIN {X 0,Y 532.634,Z 538.899,A -85,B 0,C 180,E1 25143.813,E2 25143.813} C_VEL
LIN {X 0,Y 531.769,Z 609.594,A -85,B 0,C 180,E1 25142.717,E2 25142.717} C_VEL
LIN {X 0,Y 531.043,Z 631.192,A -85,B 0,C 180,E1 25142.184,E2 25142.184} C_VEL
LIN {X 0,Y 530.19,Z 653.233,A -85,B 0,C 180,E1 25141.428,E2 25141.428} C_VEL
LIN {X 0,Y 529.207,Z 673.401,A -85,B 0,C 180,E1 25140.545,E2 25140.545} C_VEL
LIN {X 0,Y 528.048,Z 693.851,A -85,B 0,C 180,E1 25139.424,E2 25139.424} C_VEL
LIN {X 0,Y 526.793,Z 714.138,A -85,B 0,C 180,E1 25138.079,E2 25138.079} C_VEL
LIN {X 0,Y 525.57,Z 733.444,A -85,B 0,C 180,E1 25136.555,E2 25136.555} C_VEL
LIN {X 0,Y 524.426,Z 751.122,A -85,B 0,C 180,E1 25134.919,E2 25134.919} C_VEL
LIN {X 0,Y 523.333,Z 767.703,A -85,B 0,C 180,E1 25133.117,E2 25133.117} C_VEL
LIN {X 0,Y 522.409,Z 782.876,A -85,B 0,C 180,E1 25131.206,E2 25131.206} C_VEL
LIN {X 0,Y 521.626,Z 797.052,A -85,B 0,C 180,E1 25129.133,E2 25129.133} C_VEL
LIN {X 0,Y 521.011,Z 809.731,A -85,B 0,C 180,E1 25126.959,E2 25126.959} C_VEL
LIN {X 0,Y 520.563,Z 820.333,A -85,B 0,C 180,E1 25124.8,E2 25124.8} C_VEL
LIN {X 0,Y 520.243,Z 830.073,A -85,B 0,C 180,E1 25122.43,E2 25122.43} C_VEL
LIN {X 0,Y 520.066,Z 837.707,A -85,B 0,C 180,E1 25120.151,E2 25120.151} C_VEL
LIN {X 0,Y 519.97,Z 843.654,A -85,B 0,C 180,E1 25117.847,E2 25117.847} C_VEL
LIN {X 0,Y 519.926,Z 848.304,A -85,B 0,C 180,E1 25115.407,E2 25115.407} C_VEL
LIN {X 0,Y 519.916,Z 851.011,A -85,B 0,C 180,E1 25113.197,E2 25113.197} C_VEL
LIN {X 0,Y 519.904,Z 852.351,A -85,B 0,C 180,E1 25110.771,E2 25110.771} C_VEL
LIN {X 0,Y 519.898,Z 852.15,A -85,B 0,C 180,E1 25108.457,E2 25108.457} C_VEL
LIN {X 0,Y 519.906,Z 850.446,A -85,B 0,C 180,E1 25106.251,E2 25106.251} C_VEL
LIN {X 0,Y 519.93,Z 847.015,A -85,B 0,C 180,E1 25103.818,E2 25103.818} C_VEL
LIN {X 0,Y 519.982,Z 842.383,A -85,B 0,C 180,E1 25101.597,E2 25101.597} C_VEL
LIN {X 0,Y 520.095,Z 835.735,A -85,B 0,C 180,E1 25099.225,E2 25099.225} C_VEL
LIN {X 0,Y 520.314,Z 827.516,A -85,B 0,C 180,E1 25096.894,E2 25096.894} C_VEL
LIN {X 0,Y 520.635,Z 818.261,A -85,B 0,C 180,E1 25094.746,E2 25094.746} C_VEL
LIN {X 0,Y 521.11,Z 807.192,A -85,B 0,C 180,E1 25092.584,E2 25092.584} C_VEL
LIN {X 0,Y 521.751,Z 794.872,A -85,B 0,C 180,E1 25090.523,E2 25090.523} C_VEL
LIN {X 0,Y 522.52,Z 781.178,A -85,B 0,C 180,E1 25088.563,E2 25088.563} C_VEL
LIN {X 0,Y 523.465,Z 765.677,A -85,B 0,C 180,E1 25086.651,E2 25086.651} C_VEL
LIN {X 0,Y 524.555,Z 748.707,A -85,B 0,C 180,E1 25084.846,E2 25084.846} C_VEL
LIN {X 0,Y 525.763,Z 730.765,A -85,B 0,C 180,E1 25083.212,E2 25083.212} C_VEL
LIN {X 0,Y 526.962,Z 711.709,A -85,B 0,C 180,E1 25081.746,E2 25081.746} C_VEL
LIN {X 0,Y 528.155,Z 691.766,A -85,B 0,C 180,E1 25080.453,E2 25080.453} C_VEL
LIN {X 0,Y 529.272,Z 672.171,A -85,B 0,C 180,E1 25079.396,E2 25079.396} C_VEL
LIN {X 0,Y 530.226,Z 652.503,A -85,B 0,C 180,E1 25078.543,E2 25078.543} C_VEL
LIN {X 0,Y 531.093,Z 630.035,A -85,B 0,C 180,E1 25077.783,E2 25077.783} C_VEL
LIN {X 0,Y 531.789,Z 608.573,A -85,B 0,C 180,E1 25077.264,E2 25077.264} C_VEL
LIN {X 0,Y 533.603,Z 454.925,A -85,B 0,C 180,E1 25074.915,E2 25074.915} C_VEL
LIN {X 0,Y 535.054,Z 317.273,A -85,B 0,C 180,E1 25072.784,E2 25072.784} C_VEL
LIN {X 0,Y 532.409,Z 302.211,A -85,B 0,C 180,E1 25072.324,E2 25072.324} C_VEL
LIN {X 0,Y 532.66,Z 290.516,A -85,B 0,C 180,E1 25071.513,E2 25071.513} C_VEL
LIN {X 0,Y 521.731,Z 266.114,A -85,B 0,C 180,E1 25068.759,E2 25068.759} C_VEL
LIN {X 0,Y 520.581,Z 263.069,A -85,B 0,C 180,E1 25068.354,E2 25068.354} C_VEL
LIN {X 0,Y 520.587,Z 262.87,A -85,B 0,C 180,E1 25064.974,E2 25064.974} C_VEL
LIN {X 0,Y 520.546,Z 262.871,A -85,B 0,C 180,E1 25061.651,E2 25061.651} C_VEL
LIN {X 0,Y 520.542,Z 262.885,A -85,B 0,C 180,E1 25058.206,E2 25058.206} C_VEL
LIN {X 0,Y 520.586,Z 262.885,A -85,B 0,C 180,E1 25054.906,E2 25054.906} C_VEL
LIN {X 0,Y 520.532,Z 262.872,A -85,B 0,C 180,E1 25051.627,E2 25051.627} C_VEL
LIN {X 0,Y 520.527,Z 262.894,A -85,B 0,C 180,E1 25048.074,E2 25048.074} C_VEL
LIN {X 0,Y 520.576,Z 262.893,A -85,B 0,C 180,E1 25044.707,E2 25044.707} C_VEL
LIN {X 0,Y 520.526,Z 262.893,A -85,B 0,C 180,E1 25041.405,E2 25041.405} C_VEL
LIN {X 0,Y 520.513,Z 262.894,A -85,B 0,C 180,E1 25038.015,E2 25038.015} C_VEL
LIN {X 0,Y 520.574,Z 262.887,A -85,B 0,C 180,E1 25034.686,E2 25034.686} C_VEL
LIN {X 0,Y 520.512,Z 262.888,A -85,B 0,C 180,E1 25031.411,E2 25031.411} C_VEL
LIN {X 0,Y 520.516,Z 262.889,A -85,B 0,C 180,E1 25027.95,E2 25027.95} C_VEL
LIN {X 0,Y 520.578,Z 262.89,A -85,B 0,C 180,E1 25024.627,E2 25024.627} C_VEL
LIN {X 0,Y 520.526,Z 262.892,A -85,B 0,C 180,E1 25021.321,E2 25021.321} C_VEL
LIN {X 0,Y 520.528,Z 262.888,A -85,B 0,C 180,E1 25017.798,E2 25017.798} C_VEL
LIN {X 0,Y 520.586,Z 262.882,A -85,B 0,C 180,E1 25014.489,E2 25014.489} C_VEL
LIN {X 0,Y 520.544,Z 262.893,A -85,B 0,C 180,E1 25011.16,E2 25011.16} C_VEL
LIN {X 0,Y 520.538,Z 262.891,A -85,B 0,C 180,E1 25007.689,E2 25007.689} C_VEL
LIN {X 0,Y 520.59,Z 262.889,A -85,B 0,C 180,E1 25004.402,E2 25004.402} C_VEL
LIN {X 0,Y 520.565,Z 262.885,A -85,B 0,C 180,E1 25000.942,E2 25000.942} C_VEL
LIN {X 0,Y 520.55,Z 262.884,A -85,B 0,C 180,E1 24997.498,E2 24997.498} C_VEL
LIN {X 0,Y 520.58,Z 262.881,A -85,B 0,C 180,E1 24994.029,E2 24994.029} C_VEL
LIN {X 0,Y 520.587,Z 262.879,A -85,B 0,C 180,E1 24990.548,E2 24990.548} C_VEL
LIN {X 0,Y 520.564,Z 262.88,A -85,B 0,C 180,E1 24987.07,E2 24987.07} C_VEL
LIN {X 0,Y 520.569,Z 262.877,A -85,B 0,C 180,E1 24983.586,E2 24983.586} C_VEL
LIN {X 0,Y 520.579,Z 262.889,A -85,B 0,C 180,E1 24980.196,E2 24980.196} C_VEL
LIN {X 0,Y 520.582,Z 262.865,A -85,B 0,C 180,E1 24977.826,E2 24977.826} C_VEL
LIN {X 0,Y 519.58,Z 262.997,A -85,B 0,C 180,E1 24976.979,E2 24976.979} C_VEL
LIN {X 0,Y 513.153,Z 263.809,A -85,B 0,C 180,E1 24974.597,E2 24974.597} C_VEL
LIN {X 0,Y 512.639,Z 263.861,A -85,B 0,C 180,E1 24973.976,E2 24973.976} C_VEL
LIN {X 0,Y 512.638,Z 263.863,A -85,B 0,C 180,E1 24970.477,E2 24970.477} C_VEL
LIN {X 0,Y 512.672,Z 264.117,A -85,B 0,C 180,E1 24969.261,E2 24969.261} C_VEL
LIN {X 0,Y 516.606,Z 273.733,A -85,B 0,C 180,E1 24967.985,E2 24967.985} C_VEL
LIN {X 0,Y 523.82,Z 291.615,A -85,B 0,C 180,E1 24965.798,E2 24965.798} C_VEL
LIN {X 0,Y 522.058,Z 328.585,A -85,B 0,C 180,E1 24962.881,E2 24962.881} C_VEL
LIN {X 0,Y 525.05,Z 346.559,A -85,B 0,C 180,E1 24962.36,E2 24962.36} C_VEL
LIN {X 0,Y 522.226,Z 581.29,A -85,B 0,C 180,E1 24958.821,E2 24958.821} C_VEL
LIN {X 0,Y 521.729,Z 602.35,A -85,B 0,C 180,E1 24958.392,E2 24958.392} C_VEL
LIN {X 0,Y 520.937,Z 622.265,A -85,B 0,C 180,E1 24957.777,E2 24957.777} C_VEL
LIN {X 0,Y 520.021,Z 641.366,A -85,B 0,C 180,E1 24956.985,E2 24956.985} C_VEL
LIN {X 0,Y 518.892,Z 661.204,A -85,B 0,C 180,E1 24955.938,E2 24955.938} C_VEL
LIN {X 0,Y 517.744,Z 681.039,A -85,B 0,C 180,E1 24954.653,E2 24954.653} C_VEL
LIN {X 0,Y 516.714,Z 698.174,A -85,B 0,C 180,E1 24953.32,E2 24953.32} C_VEL
LIN {X 0,Y 515.716,Z 714.119,A -85,B 0,C 180,E1 24951.854,E2 24951.854} C_VEL
LIN {X 0,Y 514.733,Z 730.104,A -85,B 0,C 180,E1 24950.109,E2 24950.109} C_VEL
LIN {X 0,Y 513.891,Z 744.464,A -85,B 0,C 180,E1 24948.255,E2 24948.255} C_VEL
LIN {X 0,Y 513.218,Z 757.315,A -85,B 0,C 180,E1 24946.292,E2 24946.292} C_VEL
LIN {X 0,Y 512.695,Z 768.691,A -85,B 0,C 180,E1 24944.224,E2 24944.224} C_VEL
LIN {X 0,Y 512.324,Z 778.58,A -85,B 0,C 180,E1 24942.053,E2 24942.053} C_VEL
LIN {X 0,Y 512.107,Z 786.566,A -85,B 0,C 180,E1 24939.893,E2 24939.893} C_VEL
LIN {X 0,Y 511.985,Z 793.098,A -85,B 0,C 180,E1 24937.631,E2 24937.631} C_VEL
LIN {X 0,Y 511.923,Z 797.798,A -85,B 0,C 180,E1 24935.379,E2 24935.379} C_VEL
LIN {X 0,Y 511.91,Z 800.848,A -85,B 0,C 180,E1 24933.135,E2 24933.135} C_VEL
LIN {X 0,Y 511.91,Z 802.338,A -85,B 0,C 180,E1 24930.783,E2 24930.783} C_VEL
LIN {X 0,Y 511.9,Z 802.169,A -85,B 0,C 180,E1 24928.545,E2 24928.545} C_VEL
LIN {X 0,Y 511.91,Z 800.372,A -85,B 0,C 180,E1 24926.305,E2 24926.305} C_VEL
LIN {X 0,Y 511.942,Z 796.93,A -85,B 0,C 180,E1 24924.059,E2 24924.059} C_VEL
LIN {X 0,Y 512.01,Z 791.826,A -85,B 0,C 180,E1 24921.805,E2 24921.805} C_VEL
LIN {X 0,Y 512.141,Z 785.347,A -85,B 0,C 180,E1 24919.653,E2 24919.653} C_VEL
LIN {X 0,Y 512.389,Z 777.098,A -85,B 0,C 180,E1 24917.491,E2 24917.491} C_VEL
LIN {X 0,Y 512.783,Z 766.841,A -85,B 0,C 180,E1 24915.317,E2 24915.317} C_VEL
LIN {X 0,Y 513.294,Z 755.753,A -85,B 0,C 180,E1 24913.361,E2 24913.361} C_VEL
LIN {X 0,Y 513.997,Z 742.575,A -85,B 0,C 180,E1 24911.397,E2 24911.397} C_VEL
LIN {X 0,Y 514.862,Z 727.838,A -85,B 0,C 180,E1 24909.54,E2 24909.54} C_VEL
LIN {X 0,Y 515.802,Z 712.594,A -85,B 0,C 180,E1 24907.908,E2 24907.908} C_VEL
LIN {X 0,Y 516.859,Z 695.904,A -85,B 0,C 180,E1 24906.395,E2 24906.395} C_VEL
LIN {X 0,Y 517.983,Z 677.356,A -85,B 0,C 180,E1 24904.993,E2 24904.993} C_VEL
LIN {X 0,Y 519.184,Z 656.7,A -85,B 0,C 180,E1 24903.709,E2 24903.709} C_VEL
LIN {X 0,Y 520.182,Z 638.195,A -85,B 0,C 180,E1 24902.777,E2 24902.777} C_VEL
LIN {X 0,Y 521.082,Z 618.925,A -85,B 0,C 180,E1 24902.018,E2 24902.018} C_VEL
LIN {X 0,Y 521.81,Z 598.258,A -85,B 0,C 180,E1 24901.422,E2 24901.422} C_VEL
LIN {X 0,Y 522.302,Z 575.889,A -85,B 0,C 180,E1 24901.005,E2 24901.005} C_VEL
LIN {X 0,Y 525.032,Z 345.211,A -85,B 0,C 180,E1 24897.527,E2 24897.527} C_VEL
LIN {X 0,Y 521.999,Z 327.659,A -85,B 0,C 180,E1 24896.98,E2 24896.98} C_VEL
LIN {X 0,Y 523.752,Z 291.407,A -85,B 0,C 180,E1 24894.088,E2 24894.088} C_VEL
LIN {X 0,Y 516.723,Z 273.977,A -85,B 0,C 180,E1 24891.957,E2 24891.957} C_VEL
LIN {X 0,Y 512.691,Z 264.207,A -85,B 0,C 180,E1 24890.669,E2 24890.669} C_VEL
LIN {X 0,Y 512.628,Z 263.86,A -85,B 0,C 180,E1 24889.697,E2 24889.697} C_VEL
LIN {X 0,Y 512.642,Z 263.859,A -85,B 0,C 180,E1 24886.182,E2 24886.182} C_VEL
LIN {X 0,Y 512.632,Z 263.855,A -85,B 0,C 180,E1 24882.668,E2 24882.668} C_VEL
LIN {X 0,Y 512.649,Z 263.875,A -85,B 0,C 180,E1 24879.192,E2 24879.192} C_VEL
LIN {X 0,Y 512.64,Z 263.867,A -85,B 0,C 180,E1 24875.674,E2 24875.674} C_VEL
LIN {X 0,Y 512.638,Z 263.861,A -85,B 0,C 180,E1 24872.172,E2 24872.172} C_VEL
LIN {X 0,Y 512.623,Z 263.88,A -85,B 0,C 180,E1 24868.674,E2 24868.674} C_VEL
LIN {X 0,Y 512.64,Z 263.878,A -85,B 0,C 180,E1 24865.163,E2 24865.163} C_VEL
LIN {X 0,Y 512.649,Z 263.871,A -85,B 0,C 180,E1 24861.631,E2 24861.631} C_VEL
LIN {X 0,Y 512.619,Z 263.871,A -85,B 0,C 180,E1 24858.185,E2 24858.185} C_VEL
LIN {X 0,Y 512.607,Z 263.873,A -85,B 0,C 180,E1 24854.661,E2 24854.661} C_VEL
LIN {X 0,Y 512.642,Z 263.875,A -85,B 0,C 180,E1 24851.247,E2 24851.247} C_VEL
LIN {X 0,Y 512.632,Z 263.878,A -85,B 0,C 180,E1 24847.78,E2 24847.78} C_VEL
LIN {X 0,Y 512.593,Z 263.88,A -85,B 0,C 180,E1 24844.363,E2 24844.363} C_VEL
LIN {X 0,Y 512.609,Z 263.879,A -85,B 0,C 180,E1 24840.894,E2 24840.894} C_VEL
LIN {X 0,Y 512.632,Z 263.875,A -85,B 0,C 180,E1 24837.541,E2 24837.541} C_VEL
LIN {X 0,Y 512.581,Z 263.881,A -85,B 0,C 180,E1 24834.152,E2 24834.152} C_VEL
LIN {X 0,Y 512.586,Z 263.883,A -85,B 0,C 180,E1 24830.683,E2 24830.683} C_VEL
LIN {X 0,Y 512.633,Z 263.877,A -85,B 0,C 180,E1 24827.268,E2 24827.268} C_VEL
LIN {X 0,Y 512.571,Z 263.876,A -85,B 0,C 180,E1 24823.919,E2 24823.919} C_VEL
LIN {X 0,Y 512.573,Z 263.877,A -85,B 0,C 180,E1 24820.396,E2 24820.396} C_VEL
LIN {X 0,Y 512.633,Z 263.874,A -85,B 0,C 180,E1 24817.04,E2 24817.04} C_VEL
LIN {X 0,Y 512.594,Z 263.881,A -85,B 0,C 180,E1 24813.719,E2 24813.719} C_VEL
LIN {X 0,Y 512.587,Z 263.875,A -85,B 0,C 180,E1 24810.3,E2 24810.3} C_VEL
LIN {X 0,Y 512.644,Z 263.871,A -85,B 0,C 180,E1 24806.997,E2 24806.997} C_VEL
LIN {X 0,Y 512.606,Z 263.863,A -85,B 0,C 180,E1 24803.633,E2 24803.633} C_VEL
LIN {X 0,Y 512.601,Z 263.881,A -85,B 0,C 180,E1 24800.219,E2 24800.219} C_VEL
LIN {X 0,Y 512.644,Z 263.878,A -85,B 0,C 180,E1 24796.797,E2 24796.797} C_VEL
LIN {X 0,Y 512.635,Z 263.867,A -85,B 0,C 180,E1 24793.322,E2 24793.322} C_VEL
LIN {X 0,Y 512.658,Z 264.172,A -85,B 0,C 180,E1 24792.287,E2 24792.287} C_VEL
LIN {X 0,Y 514.038,Z 267.544,A -85,B 0,C 180,E1 24791.843,E2 24791.843} C_VEL
LIN {X 0,Y 525.654,Z 293.505,A -85,B 0,C 180,E1 24788.839,E2 24788.839} C_VEL
LIN {X 0,Y 525.951,Z 294.88,A -85,B 0,C 180,E1 24788.714,E2 24788.714} C_VEL
LIN {X 0,Y 525.757,Z 303.373,A -85,B 0,C 180,E1 24788.158,E2 24788.158} C_VEL
LIN {X 0,Y 528.651,Z 320.868,A -85,B 0,C 180,E1 24787.643,E2 24787.643} C_VEL
LIN {X 0,Y 526.324,Z 513.326,A -85,B 0,C 180,E1 24784.689,E2 24784.689} C_VEL
LIN {X 0,Y 525.049,Z 609.102,A -85,B 0,C 180,E1 24783.2,E2 24783.2} C_VEL
LIN {X 0,Y 524.283,Z 630.513,A -85,B 0,C 180,E1 24782.672,E2 24782.672} C_VEL
LIN {X 0,Y 523.346,Z 652.49,A -85,B 0,C 180,E1 24781.919,E2 24781.919} C_VEL
LIN {X 0,Y 522.312,Z 672.173,A -85,B 0,C 180,E1 24781.057,E2 24781.057} C_VEL
LIN {X 0,Y 521.076,Z 691.759,A -85,B 0,C 180,E1 24779.99,E2 24779.99} C_VEL
LIN {X 0,Y 519.71,Z 712.512,A -85,B 0,C 180,E1 24778.622,E2 24778.622} C_VEL
LIN {X 0,Y 518.439,Z 730.763,A -85,B 0,C 180,E1 24777.198,E2 24777.198} C_VEL
LIN {X 0,Y 517.11,Z 748.709,A -85,B 0,C 180,E1 24775.542,E2 24775.542} C_VEL
LIN {X 0,Y 515.9,Z 765.676,A -85,B 0,C 180,E1 24773.712,E2 24773.712} C_VEL
LIN {X 0,Y 514.847,Z 781.179,A -85,B 0,C 180,E1 24771.772,E2 24771.772} C_VEL
LIN {X 0,Y 513.942,Z 795.634,A -85,B 0,C 180,E1 24769.667,E2 24769.667} C_VEL
LIN {X 0,Y 513.204,Z 808.46,A -85,B 0,C 180,E1 24767.459,E2 24767.459} C_VEL
LIN {X 0,Y 512.664,Z 819.817,A -85,B 0,C 180,E1 24765.149,E2 24765.149} C_VEL
LIN {X 0,Y 512.314,Z 829.258,A -85,B 0,C 180,E1 24762.855,E2 24762.855} C_VEL
LIN {X 0,Y 512.102,Z 836.883,A -85,B 0,C 180,E1 24760.575,E2 24760.575} C_VEL
LIN {X 0,Y 511.987,Z 843.146,A -85,B 0,C 180,E1 24758.196,E2 24758.196} C_VEL
LIN {X 0,Y 511.928,Z 847.823,A -85,B 0,C 180,E1 24755.829,E2 24755.829} C_VEL
LIN {X 0,Y 511.911,Z 850.787,A -85,B 0,C 180,E1 24753.471,E2 24753.471} C_VEL
LIN {X 0,Y 511.912,Z 852.305,A -85,B 0,C 180,E1 24751.007,E2 24751.007} C_VEL
LIN {X 0,Y 511.903,Z 852.237,A -85,B 0,C 180,E1 24748.657,E2 24748.657} C_VEL
LIN {X 0,Y 511.906,Z 850.559,A -85,B 0,C 180,E1 24746.304,E2 24746.304} C_VEL
LIN {X 0,Y 511.932,Z 847.427,A -85,B 0,C 180,E1 24743.946,E2 24743.946} C_VEL
LIN {X 0,Y 511.989,Z 842.891,A -85,B 0,C 180,E1 24741.691,E2 24741.691} C_VEL
LIN {X 0,Y 512.111,Z 836.176,A -85,B 0,C 180,E1 24739.197,E2 24739.197} C_VEL
LIN {X 0,Y 512.35,Z 828.19,A -85,B 0,C 180,E1 24736.856,E2 24736.856} C_VEL
LIN {X 0,Y 512.71,Z 818.781,A -85,B 0,C 180,E1 24734.62,E2 24734.62} C_VEL
LIN {X 0,Y 513.277,Z 807.039,A -85,B 0,C 180,E1 24732.281,E2 24732.281} C_VEL
LIN {X 0,Y 514.021,Z 794.1,A -85,B 0,C 180,E1 24730.099,E2 24730.099} C_VEL
LIN {X 0,Y 514.965,Z 779.478,A -85,B 0,C 180,E1 24727.993,E2 24727.993} C_VEL
LIN {X 0,Y 516.047,Z 763.649,A -85,B 0,C 180,E1 24726.052,E2 24726.052} C_VEL
LIN {X 0,Y 517.263,Z 746.654,A -85,B 0,C 180,E1 24724.259,E2 24724.259} C_VEL
LIN {X 0,Y 518.57,Z 728.595,A -85,B 0,C 180,E1 24722.623,E2 24722.623} C_VEL
LIN {X 0,Y 519.899,Z 710.084,A -85,B 0,C 180,E1 24721.201,E2 24721.201} C_VEL
LIN {X 0,Y 521.139,Z 690.758,A -85,B 0,C 180,E1 24719.951,E2 24719.951} C_VEL
LIN {X 0,Y 522.418,Z 670.106,A -85,B 0,C 180,E1 24718.846,E2 24718.846} C_VEL
LIN {X 0,Y 523.437,Z 650.669,A -85,B 0,C 180,E1 24718.007,E2 24718.007} C_VEL
LIN {X 0,Y 524.335,Z 629.383,A -85,B 0,C 180,E1 24717.296,E2 24717.296} C_VEL
LIN {X 0,Y 525.067,Z 607.931,A -85,B 0,C 180,E1 24716.779,E2 24716.779} C_VEL
LIN {X 0,Y 527.873,Z 391.885,A -85,B 0,C 180,E1 24713.44,E2 24713.44} C_VEL
LIN {X 0,Y 528.496,Z 318.774,A -85,B 0,C 180,E1 24712.309,E2 24712.309} C_VEL
LIN {X 0,Y 525.655,Z 301.918,A -85,B 0,C 180,E1 24711.774,E2 24711.774} C_VEL
LIN {X 0,Y 525.872,Z 294.045,A -85,B 0,C 180,E1 24711.219,E2 24711.219} C_VEL
LIN {X 0,Y 515.297,Z 270.434,A -85,B 0,C 180,E1 24708.501,E2 24708.501} C_VEL
LIN {X 0,Y 512.673,Z 264.263,A -85,B 0,C 180,E1 24707.734,E2 24707.734} C_VEL
LIN {X 0,Y 512.648,Z 263.872,A -85,B 0,C 180,E1 24706.952,E2 24706.952} C_VEL
LIN {X 0,Y 512.625,Z 263.882,A -85,B 0,C 180,E1 24703.485,E2 24703.485} C_VEL
LIN {X 0,Y 512.6,Z 263.88,A -85,B 0,C 180,E1 24700.067,E2 24700.067} C_VEL
LIN {X 0,Y 512.637,Z 263.857,A -85,B 0,C 180,E1 24696.717,E2 24696.717} C_VEL
LIN {X 0,Y 512.614,Z 263.881,A -85,B 0,C 180,E1 24693.37,E2 24693.37} C_VEL
LIN {X 0,Y 512.586,Z 263.875,A -85,B 0,C 180,E1 24689.957,E2 24689.957} C_VEL
LIN {X 0,Y 512.632,Z 263.875,A -85,B 0,C 180,E1 24686.654,E2 24686.654} C_VEL
LIN {X 0,Y 512.601,Z 263.878,A -85,B 0,C 180,E1 24683.265,E2 24683.265} C_VEL
LIN {X 0,Y 512.573,Z 263.877,A -85,B 0,C 180,E1 24679.841,E2 24679.841} C_VEL
LIN {X 0,Y 512.616,Z 263.876,A -85,B 0,C 180,E1 24676.545,E2 24676.545} C_VEL
LIN {X 0,Y 512.582,Z 263.883,A -85,B 0,C 180,E1 24673.261,E2 24673.261} C_VEL
LIN {X 0,Y 512.573,Z 263.883,A -85,B 0,C 180,E1 24669.884,E2 24669.884} C_VEL
LIN {X 0,Y 512.639,Z 263.875,A -85,B 0,C 180,E1 24666.608,E2 24666.608} C_VEL
LIN {X 0,Y 512.591,Z 263.88,A -85,B 0,C 180,E1 24663.243,E2 24663.243} C_VEL
LIN {X 0,Y 512.586,Z 263.88,A -85,B 0,C 180,E1 24659.776,E2 24659.776} C_VEL
LIN {X 0,Y 512.639,Z 263.879,A -85,B 0,C 180,E1 24656.421,E2 24656.421} C_VEL
LIN {X 0,Y 512.611,Z 263.875,A -85,B 0,C 180,E1 24653.054,E2 24653.054} C_VEL
LIN {X 0,Y 512.597,Z 263.87,A -85,B 0,C 180,E1 24649.662,E2 24649.662} C_VEL
LIN {X 0,Y 512.642,Z 263.87,A -85,B 0,C 180,E1 24646.233,E2 24646.233} C_VEL
LIN {X 0,Y 512.64,Z 263.879,A -85,B 0,C 180,E1 24642.755,E2 24642.755} C_VEL
LIN {X 0,Y 512.61,Z 263.88,A -85,B 0,C 180,E1 24639.326,E2 24639.326} C_VEL
LIN {X 0,Y 512.627,Z 263.877,A -85,B 0,C 180,E1 24635.82,E2 24635.82} C_VEL
LIN {X 0,Y 512.647,Z 263.878,A -85,B 0,C 180,E1 24632.307,E2 24632.307} C_VEL
LIN {X 0,Y 512.635,Z 263.853,A -85,B 0,C 180,E1 24628.878,E2 24628.878} C_VEL
LIN {X 0,Y 512.625,Z 263.879,A -85,B 0,C 180,E1 24625.394,E2 24625.394} C_VEL
LIN {X 0,Y 512.647,Z 263.86,A -85,B 0,C 180,E1 24621.952,E2 24621.952} C_VEL
LIN {X 0,Y 512.641,Z 263.859,A -85,B 0,C 180,E1 24618.46,E2 24618.46} C_VEL
LIN {X 0,Y 512.638,Z 263.877,A -85,B 0,C 180,E1 24614.913,E2 24614.913} C_VEL
LIN {X 0,Y 512.639,Z 263.861,A -85,B 0,C 180,E1 24613.976,E2 24613.976} C_VEL
LIN {X 0,Y 511.647,Z 264.032,A -85,B 0,C 180,E1 24613.113,E2 24613.113} C_VEL
LIN {X 0,Y 505.169,Z 264.801,A -85,B 0,C 180,E1 24610.693,E2 24610.693} C_VEL
LIN {X 0,Y 504.704,Z 264.932,A -85,B 0,C 180,E1 24610.065,E2 24610.065} C_VEL
LIN {X 0,Y 504.823,Z 265.567,A -85,B 0,C 180,E1 24609.871,E2 24609.871} C_VEL
LIN {X 0,Y 512.777,Z 284.411,A -85,B 0,C 180,E1 24607.384,E2 24607.384} C_VEL
LIN {X 0,Y 516.912,Z 295.166,A -85,B 0,C 180,E1 24606.077,E2 24606.077} C_VEL
LIN {X 0,Y 515.202,Z 328.384,A -85,B 0,C 180,E1 24603.429,E2 24603.429} C_VEL
LIN {X 0,Y 518.484,Z 347.902,A -85,B 0,C 180,E1 24602.848,E2 24602.848} C_VEL
LIN {X 0,Y 515.526,Z 581.434,A -85,B 0,C 180,E1 24599.305,E2 24599.305} C_VEL
LIN {X 0,Y 514.984,Z 602.492,A -85,B 0,C 180,E1 24598.873,E2 24598.873} C_VEL
LIN {X 0,Y 514.152,Z 622.16,A -85,B 0,C 180,E1 24598.263,E2 24598.263} C_VEL
LIN {X 0,Y 513.191,Z 640.593,A -85,B 0,C 180,E1 24597.499,E2 24597.499} C_VEL
LIN {X 0,Y 512.095,Z 658.669,A -85,B 0,C 180,E1 24596.558,E2 24596.558} C_VEL
LIN {X 0,Y 510.839,Z 676.998,A -85,B 0,C 180,E1 24595.381,E2 24595.381} C_VEL
LIN {X 0,Y 509.489,Z 695.034,A -85,B 0,C 180,E1 24593.968,E2 24593.968} C_VEL
LIN {X 0,Y 508.137,Z 714.129,A -85,B 0,C 180,E1 24592.197,E2 24592.197} C_VEL
LIN {X 0,Y 507.055,Z 730.111,A -85,B 0,C 180,E1 24590.427,E2 24590.427} C_VEL
LIN {X 0,Y 506.177,Z 743.624,A -85,B 0,C 180,E1 24588.662,E2 24588.662} C_VEL
LIN {X 0,Y 505.412,Z 756.617,A -85,B 0,C 180,E1 24586.669,E2 24586.669} C_VEL
LIN {X 0,Y 504.823,Z 768.121,A -85,B 0,C 180,E1 24584.568,E2 24584.568} C_VEL
LIN {X 0,Y 504.423,Z 777.664,A -85,B 0,C 180,E1 24582.477,E2 24582.477} C_VEL
LIN {X 0,Y 504.156,Z 785.834,A -85,B 0,C 180,E1 24580.282,E2 24580.282} C_VEL
LIN {X 0,Y 504.007,Z 792.496,A -85,B 0,C 180,E1 24577.982,E2 24577.982} C_VEL
LIN {X 0,Y 503.935,Z 797.386,A -85,B 0,C 180,E1 24575.693,E2 24575.693} C_VEL
LIN {X 0,Y 503.907,Z 800.734,A -85,B 0,C 180,E1 24573.299,E2 24573.299} C_VEL
LIN {X 0,Y 503.912,Z 802.292,A -85,B 0,C 180,E1 24571.023,E2 24571.023} C_VEL
LIN {X 0,Y 503.906,Z 802.266,A -85,B 0,C 180,E1 24568.749,E2 24568.749} C_VEL
LIN {X 0,Y 503.907,Z 800.557,A -85,B 0,C 180,E1 24566.432,E2 24566.432} C_VEL
LIN {X 0,Y 503.936,Z 797.342,A -85,B 0,C 180,E1 24564.193,E2 24564.193} C_VEL
LIN {X 0,Y 504.01,Z 792.43,A -85,B 0,C 180,E1 24561.903,E2 24561.903} C_VEL
LIN {X 0,Y 504.162,Z 785.75,A -85,B 0,C 180,E1 24559.603,E2 24559.603} C_VEL
LIN {X 0,Y 504.45,Z 777.095,A -85,B 0,C 180,E1 24557.291,E2 24557.291} C_VEL
LIN {X 0,Y 504.892,Z 766.838,A -85,B 0,C 180,E1 24555.082,E2 24555.082} C_VEL
LIN {X 0,Y 505.461,Z 755.748,A -85,B 0,C 180,E1 24553.096,E2 24553.096} C_VEL
LIN {X 0,Y 506.246,Z 742.516,A -85,B 0,C 180,E1 24551.094,E2 24551.094} C_VEL
LIN {X 0,Y 507.202,Z 727.83,A -85,B 0,C 180,E1 24549.217,E2 24549.217} C_VEL
LIN {X 0,Y 508.238,Z 712.607,A -85,B 0,C 180,E1 24547.564,E2 24547.564} C_VEL
LIN {X 0,Y 509.575,Z 693.799,A -85,B 0,C 180,E1 24545.839,E2 24545.839} C_VEL
LIN {X 0,Y 510.869,Z 676.527,A -85,B 0,C 180,E1 24544.497,E2 24544.497} C_VEL
LIN {X 0,Y 512.137,Z 658.118,A -85,B 0,C 180,E1 24543.319,E2 24543.319} C_VEL
LIN {X 0,Y 513.228,Z 639.886,A -85,B 0,C 180,E1 24542.377,E2 24542.377} C_VEL
LIN {X 0,Y 514.25,Z 620.014,A -85,B 0,C 180,E1 24541.573,E2 24541.573} C_VEL
LIN {X 0,Y 515.038,Z 599.88,A -85,B 0,C 180,E1 24540.975,E2 24540.975} C_VEL
LIN {X 0,Y 515.57,Z 578.753,A -85,B 0,C 180,E1 24540.562,E2 24540.562} C_VEL
LIN {X 0,Y 518.476,Z 348.532,A -85,B 0,C 180,E1 24537.071,E2 24537.071} C_VEL
LIN {X 0,Y 517.941,Z 343.546,A -85,B 0,C 180,E1 24536.948,E2 24536.948} C_VEL
LIN {X 0,Y 515.129,Z 327.561,A -85,B 0,C 180,E1 24536.441,E2 24536.441} C_VEL
LIN {X 0,Y 516.834,Z 294.605,A -85,B 0,C 180,E1 24533.777,E2 24533.777} C_VEL
LIN {X 0,Y 509.162,Z 275.655,A -85,B 0,C 180,E1 24531.405,E2 24531.405} C_VEL
LIN {X 0,Y 504.753,Z 265.247,A -85,B 0,C 180,E1 24529.989,E2 24529.989} C_VEL
LIN {X 0,Y 504.71,Z 264.854,A -85,B 0,C 180,E1 24529.18,E2 24529.18} C_VEL
LIN {X 0,Y 504.695,Z 264.854,A -85,B 0,C 180,E1 24525.628,E2 24525.628} C_VEL
LIN {X 0,Y 504.705,Z 264.839,A -85,B 0,C 180,E1 24522.19,E2 24522.19} C_VEL
LIN {X 0,Y 504.691,Z 264.859,A -85,B 0,C 180,E1 24518.69,E2 24518.69} C_VEL
LIN {X 0,Y 504.702,Z 264.865,A -85,B 0,C 180,E1 24515.098,E2 24515.098} C_VEL
LIN {X 0,Y 504.702,Z 264.84,A -85,B 0,C 180,E1 24511.534,E2 24511.534} C_VEL
LIN {X 0,Y 504.708,Z 264.865,A -85,B 0,C 180,E1 24508.003,E2 24508.003} C_VEL
LIN {X 0,Y 504.68,Z 264.868,A -85,B 0,C 180,E1 24504.461,E2 24504.461} C_VEL
LIN {X 0,Y 504.685,Z 264.87,A -85,B 0,C 180,E1 24500.892,E2 24500.892} C_VEL
LIN {X 0,Y 504.708,Z 264.863,A -85,B 0,C 180,E1 24497.406,E2 24497.406} C_VEL
LIN {X 0,Y 504.692,Z 264.858,A -85,B 0,C 180,E1 24493.898,E2 24493.898} C_VEL
LIN {X 0,Y 504.663,Z 264.859,A -85,B 0,C 180,E1 24490.502,E2 24490.502} C_VEL
LIN {X 0,Y 504.688,Z 264.864,A -85,B 0,C 180,E1 24487.056,E2 24487.056} C_VEL
LIN {X 0,Y 504.696,Z 264.867,A -85,B 0,C 180,E1 24483.635,E2 24483.635} C_VEL
LIN {X 0,Y 504.65,Z 264.868,A -85,B 0,C 180,E1 24480.227,E2 24480.227} C_VEL
LIN {X 0,Y 504.655,Z 264.867,A -85,B 0,C 180,E1 24476.706,E2 24476.706} C_VEL
LIN {X 0,Y 504.706,Z 264.861,A -85,B 0,C 180,E1 24473.288,E2 24473.288} C_VEL
LIN {X 0,Y 504.649,Z 264.871,A -85,B 0,C 180,E1 24469.844,E2 24469.844} C_VEL
LIN {X 0,Y 504.63,Z 264.872,A -85,B 0,C 180,E1 24466.362,E2 24466.362} C_VEL
LIN {X 0,Y 504.679,Z 264.871,A -85,B 0,C 180,E1 24463.068,E2 24463.068} C_VEL
LIN {X 0,Y 504.651,Z 264.866,A -85,B 0,C 180,E1 24459.713,E2 24459.713} C_VEL
LIN {X 0,Y 504.639,Z 264.869,A -85,B 0,C 180,E1 24456.256,E2 24456.256} C_VEL
LIN {X 0,Y 504.688,Z 264.867,A -85,B 0,C 180,E1 24452.893,E2 24452.893} C_VEL
LIN {X 0,Y 504.674,Z 264.848,A -85,B 0,C 180,E1 24449.519,E2 24449.519} C_VEL
LIN {X 0,Y 504.652,Z 264.872,A -85,B 0,C 180,E1 24446.112,E2 24446.112} C_VEL
LIN {X 0,Y 504.685,Z 264.847,A -85,B 0,C 180,E1 24442.683,E2 24442.683} C_VEL
LIN {X 0,Y 504.697,Z 264.849,A -85,B 0,C 180,E1 24439.324,E2 24439.324} C_VEL
LIN {X 0,Y 504.666,Z 264.869,A -85,B 0,C 180,E1 24435.94,E2 24435.94} C_VEL
LIN {X 0,Y 504.749,Z 265.13,A -85,B 0,C 180,E1 24432.991,E2 24432.991} C_VEL
LIN {X 0,Y 506.095,Z 268.512,A -85,B 0,C 180,E1 24432.531,E2 24432.531} C_VEL
LIN {X 0,Y 514.69,Z 287.504,A -85,B 0,C 180,E1 24430.23,E2 24430.23} C_VEL
LIN {X 0,Y 519.122,Z 298.182,A -85,B 0,C 180,E1 24429.036,E2 24429.036} C_VEL
LIN {X 0,Y 519.041,Z 303.665,A -85,B 0,C 180,E1 24428.685,E2 24428.685} C_VEL
LIN {X 0,Y 522.08,Z 322.345,A -85,B 0,C 180,E1 24428.125,E2 24428.125} C_VEL
LIN {X 0,Y 519.363,Z 540.553,A -85,B 0,C 180,E1 24424.772,E2 24424.772} C_VEL
LIN {X 0,Y 518.341,Z 609.593,A -85,B 0,C 180,E1 24423.676,E2 24423.676} C_VEL
LIN {X 0,Y 517.514,Z 630.927,A -85,B 0,C 180,E1 24423.14,E2 24423.14} C_VEL
LIN {X 0,Y 516.464,Z 653.227,A -85,B 0,C 180,E1 24422.363,E2 24422.363} C_VEL
LIN {X 0,Y 515.307,Z 673.396,A -85,B 0,C 180,E1 24421.462,E2 24421.462} C_VEL
LIN {X 0,Y 513.906,Z 693.765,A -85,B 0,C 180,E1 24420.323,E2 24420.323} C_VEL
LIN {X 0,Y 512.48,Z 713.32,A -85,B 0,C 180,E1 24419,E2 24419} C_VEL
LIN {X 0,Y 511.085,Z 731.434,A -85,B 0,C 180,E1 24417.559,E2 24417.559} C_VEL
LIN {X 0,Y 509.65,Z 749.298,A -85,B 0,C 180,E1 24415.882,E2 24415.882} C_VEL
LIN {X 0,Y 508.389,Z 765.225,A -85,B 0,C 180,E1 24414.139,E2 24414.139} C_VEL
LIN {X 0,Y 507.248,Z 780.33,A -85,B 0,C 180,E1 24412.238,E2 24412.238} C_VEL
LIN {X 0,Y 506.224,Z 794.87,A -85,B 0,C 180,E1 24410.1,E2 24410.1} C_VEL
LIN {X 0,Y 505.419,Z 807.541,A -85,B 0,C 180,E1 24407.909,E2 24407.909} C_VEL
LIN {X 0,Y 504.787,Z 819.301,A -85,B 0,C 180,E1 24405.509,E2 24405.509} C_VEL
LIN {X 0,Y 504.382,Z 828.851,A -85,B 0,C 180,E1 24403.177,E2 24403.177} C_VEL
LIN {X 0,Y 504.129,Z 836.53,A -85,B 0,C 180,E1 24400.86,E2 24400.86} C_VEL
LIN {X 0,Y 503.994,Z 843.146,A -85,B 0,C 180,E1 24398.327,E2 24398.327} C_VEL
LIN {X 0,Y 503.93,Z 847.823,A -85,B 0,C 180,E1 24395.922,E2 24395.922} C_VEL
LIN {X 0,Y 503.909,Z 850.787,A -85,B 0,C 180,E1 24393.526,E2 24393.526} C_VEL
LIN {X 0,Y 503.912,Z 852.305,A -85,B 0,C 180,E1 24391.023,E2 24391.023} C_VEL
LIN {X 0,Y 503.906,Z 852.259,A -85,B 0,C 180,E1 24388.749,E2 24388.749} C_VEL
LIN {X 0,Y 503.907,Z 850.673,A -85,B 0,C 180,E1 24386.36,E2 24386.36} C_VEL
LIN {X 0,Y 503.933,Z 847.633,A -85,B 0,C 180,E1 24383.964,E2 24383.964} C_VEL
LIN {X 0,Y 503.993,Z 842.891,A -85,B 0,C 180,E1 24381.558,E2 24381.558} C_VEL
LIN {X 0,Y 504.137,Z 836.176,A -85,B 0,C 180,E1 24379.024,E2 24379.024} C_VEL
LIN {X 0,Y 504.4,Z 828.429,A -85,B 0,C 180,E1 24376.707,E2 24376.707} C_VEL
LIN {X 0,Y 504.816,Z 818.782,A -85,B 0,C 180,E1 24374.374,E2 24374.374} C_VEL
LIN {X 0,Y 505.441,Z 807.189,A -85,B 0,C 180,E1 24372.026,E2 24372.026} C_VEL
LIN {X 0,Y 506.224,Z 794.869,A -85,B 0,C 180,E1 24369.9,E2 24369.9} C_VEL
LIN {X 0,Y 507.248,Z 780.33,A -85,B 0,C 180,E1 24367.762,E2 24367.762} C_VEL
LIN {X 0,Y 508.393,Z 765.169,A -85,B 0,C 180,E1 24365.854,E2 24365.854} C_VEL
LIN {X 0,Y 509.746,Z 748.1,A -85,B 0,C 180,E1 24363.999,E2 24363.999} C_VEL
LIN {X 0,Y 511.141,Z 730.764,A -85,B 0,C 180,E1 24362.381,E2 24362.381} C_VEL
LIN {X 0,Y 512.575,Z 712.163,A -85,B 0,C 180,E1 24360.914,E2 24360.914} C_VEL
LIN {X 0,Y 514.036,Z 691.759,A -85,B 0,C 180,E1 24359.557,E2 24359.557} C_VEL
LIN {X 0,Y 515.383,Z 672.177,A -85,B 0,C 180,E1 24358.478,E2 24358.478} C_VEL
LIN {X 0,Y 516.541,Z 651.759,A -85,B 0,C 180,E1 24357.577,E2 24357.577} C_VEL
LIN {X 0,Y 517.562,Z 629.955,A -85,B 0,C 180,E1 24356.832,E2 24356.832} C_VEL
LIN {X 0,Y 518.361,Z 608.681,A -85,B 0,C 180,E1 24356.307,E2 24356.307} C_VEL
LIN {X 0,Y 519.989,Z 493.412,A -85,B 0,C 180,E1 24354.504,E2 24354.504} C_VEL
LIN {X 0,Y 521.999,Z 320.635,A -85,B 0,C 180,E1 24351.84,E2 24351.84} C_VEL
LIN {X 0,Y 518.936,Z 302.49,A -85,B 0,C 180,E1 24351.263,E2 24351.263} C_VEL
LIN {X 0,Y 519.096,Z 297.576,A -85,B 0,C 180,E1 24350.917,E2 24350.917} C_VEL
LIN {X 0,Y 508.132,Z 272.784,A -85,B 0,C 180,E1 24348.01,E2 24348.01} C_VEL
LIN {X 0,Y 504.777,Z 265.3,A -85,B 0,C 180,E1 24347.049,E2 24347.049} C_VEL
LIN {X 0,Y 504.679,Z 264.852,A -85,B 0,C 180,E1 24346.415,E2 24346.415} C_VEL
LIN {X 0,Y 504.71,Z 264.859,A -85,B 0,C 180,E1 24342.959,E2 24342.959} C_VEL
LIN {X 0,Y 504.678,Z 264.869,A -85,B 0,C 180,E1 24339.491,E2 24339.491} C_VEL
LIN {X 0,Y 504.656,Z 264.855,A -85,B 0,C 180,E1 24336.046,E2 24336.046} C_VEL
LIN {X 0,Y 504.688,Z 264.853,A -85,B 0,C 180,E1 24332.606,E2 24332.606} C_VEL
LIN {X 0,Y 504.672,Z 264.863,A -85,B 0,C 180,E1 24329.298,E2 24329.298} C_VEL
LIN {X 0,Y 504.643,Z 264.87,A -85,B 0,C 180,E1 24325.908,E2 24325.908} C_VEL
LIN {X 0,Y 504.674,Z 264.868,A -85,B 0,C 180,E1 24322.48,E2 24322.48} C_VEL
LIN {X 0,Y 504.67,Z 264.863,A -85,B 0,C 180,E1 24319.089,E2 24319.089} C_VEL
LIN {X 0,Y 504.627,Z 264.864,A -85,B 0,C 180,E1 24315.75,E2 24315.75} C_VEL
LIN {X 0,Y 504.658,Z 264.865,A -85,B 0,C 180,E1 24312.355,E2 24312.355} C_VEL
LIN {X 0,Y 504.669,Z 264.873,A -85,B 0,C 180,E1 24309.005,E2 24309.005} C_VEL
LIN {X 0,Y 504.638,Z 264.871,A -85,B 0,C 180,E1 24305.685,E2 24305.685} C_VEL
LIN {X 0,Y 504.673,Z 264.867,A -85,B 0,C 180,E1 24302.271,E2 24302.271} C_VEL
LIN {X 0,Y 504.676,Z 264.865,A -85,B 0,C 180,E1 24298.978,E2 24298.978} C_VEL
LIN {X 0,Y 504.65,Z 264.87,A -85,B 0,C 180,E1 24295.568,E2 24295.568} C_VEL
LIN {X 0,Y 504.682,Z 264.868,A -85,B 0,C 180,E1 24292.119,E2 24292.119} C_VEL
LIN {X 0,Y 504.703,Z 264.863,A -85,B 0,C 180,E1 24288.689,E2 24288.689} C_VEL
LIN {X 0,Y 504.664,Z 264.862,A -85,B 0,C 180,E1 24285.309,E2 24285.309} C_VEL
LIN {X 0,Y 504.676,Z 264.86,A -85,B 0,C 180,E1 24281.758,E2 24281.758} C_VEL
LIN {X 0,Y 504.711,Z 264.858,A -85,B 0,C 180,E1 24278.256,E2 24278.256} C_VEL
LIN {X 0,Y 504.699,Z 264.866,A -85,B 0,C 180,E1 24274.79,E2 24274.79} C_VEL
LIN {X 0,Y 504.678,Z 264.869,A -85,B 0,C 180,E1 24271.351,E2 24271.351} C_VEL
LIN {X 0,Y 504.704,Z 264.844,A -85,B 0,C 180,E1 24267.931,E2 24267.931} C_VEL
LIN {X 0,Y 504.704,Z 264.857,A -85,B 0,C 180,E1 24264.378,E2 24264.378} C_VEL
LIN {X 0,Y 504.707,Z 264.863,A -85,B 0,C 180,E1 24260.767,E2 24260.767} C_VEL
LIN {X 0,Y 504.69,Z 264.843,A -85,B 0,C 180,E1 24257.193,E2 24257.193} C_VEL
LIN {X 0,Y 504.704,Z 264.845,A -85,B 0,C 180,E1 24253.689,E2 24253.689} C_VEL
LIN {X 0,Y 504.692,Z 264.848,A -85,B 0,C 180,E1 24250.228,E2 24250.228} C_VEL
LIN {X 0,Y 504.704,Z 264.932,A -85,B 0,C 180,E1 24250.065,E2 24250.065} C_VEL
LIN {X 0,Y 505.835,Z 265.78,A -85,B 0,C 180,E1 24249.744,E2 24249.744} C_VEL
LIN {X 0,Y 507.928,Z 268.657,A -85,B 0,C 180,E1 24249.262,E2 24249.262} C_VEL
LIN {X 0,Y 508.546,Z 272.719,A -85,B 0,C 180,E1 24248.831,E2 24248.831} C_VEL
LIN {X 0,Y 508.144,Z 279.549,A -85,B 0,C 180,E1 24248.294,E2 24248.294} C_VEL
LIN {X 0,Y 506.787,Z 287.412,A -85,B 0,C 180,E1 24247.678,E2 24247.678} C_VEL
LIN {X 0,Y 507.172,Z 290.873,A -85,B 0,C 180,E1 24247.316,E2 24247.316} C_VEL
LIN {X 0,Y 510.016,Z 298.716,A -85,B 0,C 180,E1 24246.364,E2 24246.364} C_VEL
LIN {X 0,Y 508.383,Z 328.138,A -85,B 0,C 180,E1 24243.995,E2 24243.995} C_VEL
LIN {X 0,Y 511.957,Z 349.256,A -85,B 0,C 180,E1 24243.348,E2 24243.348} C_VEL
LIN {X 0,Y 508.868,Z 581.962,A -85,B 0,C 180,E1 24239.798,E2 24239.798} C_VEL
LIN {X 0,Y 508.293,Z 603.077,A -85,B 0,C 180,E1 24239.36,E2 24239.36} C_VEL
LIN {X 0,Y 507.393,Z 622.818,A -85,B 0,C 180,E1 24238.738,E2 24238.738} C_VEL
LIN {X 0,Y 506.343,Z 641.153,A -85,B 0,C 180,E1 24237.967,E2 24237.967} C_VEL
LIN {X 0,Y 505.069,Z 660.113,A -85,B 0,C 180,E1 24236.957,E2 24236.957} C_VEL
LIN {X 0,Y 503.705,Z 678.248,A -85,B 0,C 180,E1 24235.766,E2 24235.766} C_VEL
LIN {X 0,Y 502.24,Z 696.162,A -85,B 0,C 180,E1 24234.336,E2 24234.336} C_VEL
LIN {X 0,Y 500.819,Z 712.937,A -85,B 0,C 180,E1 24232.726,E2 24232.726} C_VEL
LIN {X 0,Y 499.554,Z 728.185,A -85,B 0,C 180,E1 24230.993,E2 24230.993} C_VEL
LIN {X 0,Y 498.486,Z 742.784,A -85,B 0,C 180,E1 24229.083,E2 24229.083} C_VEL
LIN {X 0,Y 497.628,Z 755.92,A -85,B 0,C 180,E1 24227.058,E2 24227.058} C_VEL
LIN {X 0,Y 496.962,Z 767.55,A -85,B 0,C 180,E1 24224.923,E2 24224.923} C_VEL
LIN {X 0,Y 496.509,Z 777.206,A -85,B 0,C 180,E1 24222.798,E2 24222.798} C_VEL
LIN {X 0,Y 496.189,Z 785.836,A -85,B 0,C 180,E1 24220.449,E2 24220.449} C_VEL
LIN {X 0,Y 496.019,Z 792.498,A -85,B 0,C 180,E1 24218.111,E2 24218.111} C_VEL
LIN {X 0,Y 495.941,Z 797.387,A -85,B 0,C 180,E1 24215.785,E2 24215.785} C_VEL
LIN {X 0,Y 495.907,Z 800.734,A -85,B 0,C 180,E1 24213.352,E2 24213.352} C_VEL
LIN {X 0,Y 495.912,Z 802.292,A -85,B 0,C 180,E1 24211.04,E2 24211.04} C_VEL
LIN {X 0,Y 495.905,Z 802.266,A -85,B 0,C 180,E1 24208.729,E2 24208.729} C_VEL
LIN {X 0,Y 495.908,Z 800.585,A -85,B 0,C 180,E1 24206.405,E2 24206.405} C_VEL
LIN {X 0,Y 495.942,Z 797.34,A -85,B 0,C 180,E1 24204.099,E2 24204.099} C_VEL
LIN {X 0,Y 496.024,Z 792.428,A -85,B 0,C 180,E1 24201.772,E2 24201.772} C_VEL
LIN {X 0,Y 496.196,Z 785.748,A -85,B 0,C 180,E1 24199.434,E2 24199.434} C_VEL
LIN {X 0,Y 496.512,Z 777.093,A -85,B 0,C 180,E1 24197.084,E2 24197.084} C_VEL
LIN {X 0,Y 497.006,Z 766.835,A -85,B 0,C 180,E1 24194.84,E2 24194.84} C_VEL
LIN {X 0,Y 497.639,Z 755.742,A -85,B 0,C 180,E1 24192.822,E2 24192.822} C_VEL
LIN {X 0,Y 498.501,Z 742.563,A -85,B 0,C 180,E1 24190.796,E2 24190.796} C_VEL
LIN {X 0,Y 499.647,Z 726.921,A -85,B 0,C 180,E1 24188.765,E2 24188.765} C_VEL
LIN {X 0,Y 500.991,Z 710.872,A -85,B 0,C 180,E1 24186.973,E2 24186.973} C_VEL
LIN {X 0,Y 502.381,Z 694.345,A -85,B 0,C 180,E1 24185.421,E2 24185.421} C_VEL
LIN {X 0,Y 503.744,Z 677.785,A -85,B 0,C 180,E1 24184.109,E2 24184.109} C_VEL
LIN {X 0,Y 505.196,Z 658.574,A -85,B 0,C 180,E1 24182.859,E2 24182.859} C_VEL
LIN {X 0,Y 506.387,Z 640.418,A -85,B 0,C 180,E1 24181.907,E2 24181.907} C_VEL
LIN {X 0,Y 507.509,Z 620.437,A -85,B 0,C 180,E1 24181.088,E2 24181.088} C_VEL
LIN {X 0,Y 508.357,Z 600.318,A -85,B 0,C 180,E1 24180.483,E2 24180.483} C_VEL
LIN {X 0,Y 508.919,Z 579.204,A -85,B 0,C 180,E1 24180.067,E2 24180.067} C_VEL
LIN {X 0,Y 511.941,Z 348.025,A -85,B 0,C 180,E1 24176.54,E2 24176.54} C_VEL
LIN {X 0,Y 508.306,Z 327.247,A -85,B 0,C 180,E1 24175.869,E2 24175.869} C_VEL
LIN {X 0,Y 510.013,Z 298.136,A -85,B 0,C 180,E1 24173.494,E2 24173.494} C_VEL
LIN {X 0,Y 502.607,Z 279.862,A -85,B 0,C 180,E1 24171.163,E2 24171.163} C_VEL
LIN {X 0,Y 496.836,Z 266.292,A -85,B 0,C 180,E1 24169.284,E2 24169.284} C_VEL
LIN {X 0,Y 496.764,Z 265.855,A -85,B 0,C 180,E1 24168.688,E2 24168.688} C_VEL
LIN {X 0,Y 496.764,Z 265.852,A -85,B 0,C 180,E1 24165.053,E2 24165.053} C_VEL
LIN {X 0,Y 496.76,Z 265.833,A -85,B 0,C 180,E1 24161.468,E2 24161.468} C_VEL
LIN {X 0,Y 496.762,Z 265.833,A -85,B 0,C 180,E1 24157.872,E2 24157.872} C_VEL
